//     Standard Inputs/Fix04.N90_STAT/Channel_4/Channel_Error <-> DPO Inputs Channel 4/Channel Error
//     Standard Inputs/Fix04.N90_STAT/Channel_1/Error_Up <-> DPO Inputs Channel 1/Error Up
//     Standard Inputs/Fix04.N90_STAT/Channel_2/Error_Up <-> DPO Inputs Channel 2/Error Up
//     Standard Inputs/Fix04.N90_STAT/Channel_3/Error_Up <-> DPO Inputs Channel 3/Error Up
//     Standard Inputs/Fix04.N90_STAT/Channel_4/Error_Up <-> DPO Inputs Channel 4/Error Up
//     Standard Inputs/Fix04.N90_STAT/Channel_1/Error_Us <-> DPO Inputs Channel 1/Error Us
//     Standard Inputs/Fix04.N90_STAT/Channel_2/Error_Us <-> DPO Inputs Channel 2/Error Us
//     Standard Inputs/Fix04.N90_STAT/Channel_3/Error_Us <-> DPO Inputs Channel 3/Error Us
//     Standard Inputs/Fix04.N90_STAT/Channel_4/Error_Us <-> DPO Inputs Channel 4/Error Us
//     Standard Inputs/Fix04.N90_STAT/Channel_1/Status_Up <-> DPO Inputs Channel 1/Status Up
//     Standard Inputs/Fix04.N90_STAT/Channel_2/Status_Up <-> DPO Inputs Channel 2/Status Up
//     Standard Inputs/Fix04.N90_STAT/Channel_3/Status_Up <-> DPO Inputs Channel 3/Status Up
//     Standard Inputs/Fix04.N90_STAT/Channel_4/Status_Up <-> DPO Inputs Channel 4/Status Up
//     Standard Inputs/Fix04.N90_STAT/Channel_1/Status_Us <-> DPO Inputs Channel 1/Status Us
//     Standard Inputs/Fix04.N90_STAT/Channel_2/Status_Us <-> DPO Inputs Channel 2/Status Us
//     Standard Inputs/Fix04.N90_STAT/Channel_3/Status_Us <-> DPO Inputs Channel 3/Status Us
//     Standard Inputs/Fix04.N90_STAT/Channel_4/Status_Us <-> DPO Inputs Channel 4/Status Us
//     Standard Inputs/Fix04.N90_STAT/Channel_1/SyncError <-> DPO Inputs Channel 1/Sync error
//     Standard Inputs/Fix04.N90_STAT/Channel_2/SyncError <-> DPO Inputs Channel 2/Sync error
//     Standard Inputs/Fix04.N90_STAT/Channel_3/SyncError <-> DPO Inputs Channel 3/Sync error
//     Standard Inputs/Fix04.N90_STAT/Channel_4/SyncError <-> DPO Inputs Channel 4/Sync error
//     Standard Inputs/Fix04.N90_STAT/Channel_1/TxPDO_State <-> DPO Inputs Channel 1/TxPDO State
//     Standard Inputs/Fix04.N90_STAT/Channel_2/TxPDO_State <-> DPO Inputs Channel 2/TxPDO State
//     Standard Inputs/Fix04.N90_STAT/Channel_3/TxPDO_State <-> DPO Inputs Channel 3/TxPDO State
//     Standard Inputs/Fix04.N90_STAT/Channel_4/TxPDO_State <-> DPO Inputs Channel 4/TxPDO State
//     Standard Inputs/Fix04.N90_STAT/Channel_1/TxPDO_Toggle <-> DPO Inputs Channel 1/TxPDO Toggle
//     Standard Inputs/Fix04.N90_STAT/Channel_2/TxPDO_Toggle <-> DPO Inputs Channel 2/TxPDO Toggle
//     Standard Inputs/Fix04.N90_STAT/Channel_3/TxPDO_Toggle <-> DPO Inputs Channel 3/TxPDO Toggle
//     Standard Inputs/Fix04.N90_STAT/Channel_4/TxPDO_Toggle <-> DPO Inputs Channel 4/TxPDO Toggle
//     Standard Inputs/Fix04.N90_STAT/Channel_1/Warning_Up <-> DPO Inputs Channel 1/Warning Up
//     Standard Inputs/Fix04.N90_STAT/Channel_2/Warning_Up <-> DPO Inputs Channel 2/Warning Up
//     Standard Inputs/Fix04.N90_STAT/Channel_3/Warning_Up <-> DPO Inputs Channel 3/Warning Up
//     Standard Inputs/Fix04.N90_STAT/Channel_4/Warning_Up <-> DPO Inputs Channel 4/Warning Up
//     Standard Inputs/Fix04.N90_STAT/Channel_1/Warning_Us <-> DPO Inputs Channel 1/Warning Us
//     Standard Inputs/Fix04.N90_STAT/Channel_2/Warning_Us <-> DPO Inputs Channel 2/Warning Us
//     Standard Inputs/Fix04.N90_STAT/Channel_3/Warning_Us <-> DPO Inputs Channel 3/Warning Us
//     Standard Inputs/Fix04.N90_STAT/Channel_4/Warning_Us <-> DPO Inputs Channel 4/Warning Us
//     Standard Inputs/Fix04.N90_STAT/Device/Global_Error_Bit <-> DPO Inputs Device/Global Error Bit
//     Standard Inputs/Fix04.N90_STAT/Device/Reset_Input <-> DPO Inputs Device/Reset Input
//     Standard Inputs/Fix04.N90_STAT/Device/Temperature_Error <-> DPO Inputs Device/Temperature Error
//     Standard Inputs/Fix04.N90_STAT/Device/Temperature_Warning <-> DPO Inputs Device/Temperature Warning
//     Standard Inputs/Fix04.N90_STAT/Device/TxPDO_State <-> DPO Inputs Device/TxPDO State
//     Standard Inputs/Fix04.N90_STAT/Device/TxPDO_Toggle <-> DPO Inputs Device/TxPDO Toggle
//     Standard Inputs/Fix04.N90_STAT/Device/Up_Error <-> DPO Inputs Device/Up Error
//     Standard Inputs/Fix04.N90_STAT/Device/Up_Warning <-> DPO Inputs Device/Up Warning
//     Standard Inputs/Fix04.N90_STAT/Device/Us_Error <-> DPO Inputs Device/Us Error
//     Standard Inputs/Fix04.N90_STAT/Device/Us_Warning <-> DPO Inputs Device/Us Warning
//     Standard Inputs/Fix04.N90_STAT/InfoData/AdsAddr <-> InfoData/AdsAddr
//     Standard Inputs/Fix04.N90_STAT/InfoData/State <-> InfoData/State
//     Standard Inputs/Fix04.N90_STAT/Wc_State <-> WcState/WcState
//     Standard Outputs/Fix04.N90_CMD/Channel1/Output_Up <-> DPO Outputs Channel 1/Output Up
//     Standard Outputs/Fix04.N90_CMD/Channel2/Output_Up <-> DPO Outputs Channel 2/Output Up
//     Standard Outputs/Fix04.N90_CMD/Channel3/Output_Up <-> DPO Outputs Channel 3/Output Up
//     Standard Outputs/Fix04.N90_CMD/Channel4/Output_Up <-> DPO Outputs Channel 4/Output Up
//     Standard Outputs/Fix04.N90_CMD/Channel1/Output_Us <-> DPO Outputs Channel 1/Output Us
//     Standard Outputs/Fix04.N90_CMD/Channel2/Output_Us <-> DPO Outputs Channel 2/Output Us
//     Standard Outputs/Fix04.N90_CMD/Channel3/Output_Us <-> DPO Outputs Channel 3/Output Us
//     Standard Outputs/Fix04.N90_CMD/Channel4/Output_Us <-> DPO Outputs Channel 4/Output Us
//     Standard Outputs/Fix04.N90_CMD/Channel1/Reset_Up <-> DPO Outputs Channel 1/Reset Up
//     Standard Outputs/Fix04.N90_CMD/Channel2/Reset_Up <-> DPO Outputs Channel 2/Reset Up
//     Standard Outputs/Fix04.N90_CMD/Channel3/Reset_Up <-> DPO Outputs Channel 3/Reset Up
//     Standard Outputs/Fix04.N90_CMD/Channel4/Reset_Up <-> DPO Outputs Channel 4/Reset Up
//     Standard Outputs/Fix04.N90_CMD/Channel1/Reset_Us <-> DPO Outputs Channel 1/Reset Us
//     Standard Outputs/Fix04.N90_CMD/Channel2/Reset_Us <-> DPO Outputs Channel 2/Reset Us
//     Standard Outputs/Fix04.N90_CMD/Channel3/Reset_Us <-> DPO Outputs Channel 3/Reset Us
//     Standard Outputs/Fix04.N90_CMD/Channel4/Reset_Us <-> DPO Outputs Channel 4/Reset Us
//     Standard Outputs/Fix04.N90_CMD/Device/Enable_Control_Via_Fieldbus <-> DPO Outputs Device/Enable Control Via Fieldbus
//     Standard Outputs/Fix04.N90_CMD/Device/Global_Reset <-> DPO Outputs Device/Global Reset
//   SODG11_SSCC610_2403701_PLC/SODG11_SSCC610_2403701_PLC Instance <-> EtherCAT Master (EtherCAT)/IC02.T01 (EK1100)/IC02.T16 (EK1122)/Fix04.N98  (EP2328-0002)
//     Standard Inputs/Fix04.N98.I <-> Channel 1/Input
//     Standard Inputs/Fix04.N98.I @bit 1 <-> Channel 2/Input
//     Standard Inputs/Fix04.N98.I @bit 2 <-> Channel 3/Input
//     Standard Inputs/Fix04.N98.I @bit 3 <-> Channel 4/Input
//     Standard Inputs/Fix04.N98.State <-> InfoData/State
//     Standard Inputs/Fix04.N98.WC_State <-> WcState/WcState
//     Standard Outputs/Fix04.N98.Q <-> Channel 5/Output
//     Standard Outputs/Fix04.N98.Q @bit 1 <-> Channel 6/Output
//     Standard Outputs/Fix04.N98.Q @bit 2 <-> Channel 7/Output
//     Standard Outputs/Fix04.N98.Q @bit 3 <-> Channel 8/Output
//   SODG11_SSCC610_2403701_PLC/SODG11_SSCC610_2403701_PLC Instance <-> EtherCAT Master (EtherCAT)/IC03.T01 (EK1100)
//     Standard Inputs/MAIN.IC03.T01/InfoData/State <-> InfoData/State
//   SODG11_SSCC610_2403701_PLC/SODG11_SSCC610_2403701_PLC Instance <-> EtherCAT Master (EtherCAT)/IC03.T01 (EK1100)/IC03.T02 (EL6900)
//     Standard Inputs/MAIN.IC03.T02_STAT/Device_Info_Data/Project_CRC <-> Device Info Data/Project CRC
//     Standard Inputs/MAIN.IC03.T02_STAT/FBs_FB_ERR <-> StandardInputs/Standard Out Var 26
//     Standard Inputs/MAIN.IC03.T02_STAT/FBs_FB_ERR @bit 8 <-> StandardInputs/Standard Out Var 27
//     Standard Inputs/MAIN.IC03.T02_STAT/FBs_FB_ERR @bit 16 <-> StandardInputs/Standard Out Var 28
//     Standard Inputs/MAIN.IC03.T02_STAT/FBs_FB_ERR @bit 17 <-> StandardInputs/Standard Out Var 29
//     Standard Inputs/MAIN.IC03.T02_STAT/InfoData/AdsAddr/netId <-> InfoData/AdsAddr/netId
//     Standard Inputs/MAIN.IC03.T02_STAT/InfoData/AdsAddr/port <-> InfoData/AdsAddr/port
//     Standard Inputs/MAIN.IC03.T02_STAT/InfoData/State <-> InfoData/State
//     Standard Inputs/MAIN.IC03.T02_STAT/SGs_COM_ERR <-> StandardInputs/Standard Out Var 17
//     Standard Inputs/MAIN.IC03.T02_STAT/SGs_COM_ERR @bit 1 <-> StandardInputs/Standard Out Var 20
//     Standard Inputs/MAIN.IC03.T02_STAT/SGs_FB_ERR <-> StandardInputs/Standard Out Var 16
//     Standard Inputs/MAIN.IC03.T02_STAT/SGs_FB_ERR @bit 1 <-> StandardInputs/Standard Out Var 19
//     Standard Inputs/MAIN.IC03.T02_STAT/SGs_OUT_ERR <-> StandardInputs/Standard Out Var 18
//     Standard Inputs/MAIN.IC03.T02_STAT/SGs_OUT_ERR @bit 1 <-> StandardInputs/Standard Out Var 25
//     Standard Inputs/MAIN.IC03.T09/Q <-> StandardInputs/Standard Out Var 21
//     Standard Inputs/MAIN.IC03.T10/Q <-> StandardInputs/Standard Out Var 23
//     Standard Inputs/MAIN.IC03.T09/Q @bit 1 <-> StandardInputs/Standard Out Var 22
//     Standard Inputs/MAIN.IC03.T10/Q @bit 1 <-> StandardInputs/Standard Out Var 24
//     Standard Outputs/MAIN.IC03.T02_CMD/FBs_ControlPowerPB <-> StandardOutputs/Standard In Var 14
//     Standard Outputs/MAIN.IC03.T02_CMD/SGs_ERRAck <-> StandardOutputs/Standard In Var 11
//     Standard Outputs/MAIN.IC03.T02_CMD/SGs_ERRAck <-> StandardOutputs/Standard In Var 13
//     Standard Outputs/MAIN.IC03.T02_CMD/SGs_RUNSTOP <-> StandardOutputs/Standard In Var 10
//     Standard Outputs/MAIN.IC03.T02_CMD/SGs_RUNSTOP <-> StandardOutputs/Standard In Var 12
//   SODG11_SSCC610_2403701_PLC/SODG11_SSCC610_2403701_PLC Instance <-> EtherCAT Master (EtherCAT)/IC03.T01 (EK1100)/IC03.T03 (EL1904)
//     Standard Inputs/MAIN.IC03.T03/I <-> Module 1 (FSOES)/TxPDO/FSOE/InputChannel1
//     Standard Inputs/MAIN.IC03.T03/I @bit 1 <-> Module 1 (FSOES)/TxPDO/FSOE/InputChannel2
//     Standard Inputs/MAIN.IC03.T03/I @bit 2 <-> Module 1 (FSOES)/TxPDO/FSOE/InputChannel3
//     Standard Inputs/MAIN.IC03.T03/I @bit 3 <-> Module 1 (FSOES)/TxPDO/FSOE/InputChannel4
//     Standard Inputs/MAIN.IC03.T03/InfoData/State <-> InfoData/State
//   SODG11_SSCC610_2403701_PLC/SODG11_SSCC610_2403701_PLC Instance <-> EtherCAT Master (EtherCAT)/IC03.T01 (EK1100)/IC03.T04 (EL1904)
//     Standard Inputs/MAIN.IC03.T04/I <-> Module 1 (FSOES)/TxPDO/FSOE/InputChannel1
//     Standard Inputs/MAIN.IC03.T04/I @bit 1 <-> Module 1 (FSOES)/TxPDO/FSOE/InputChannel2
//     Standard Inputs/MAIN.IC03.T04/I @bit 2 <-> Module 1 (FSOES)/TxPDO/FSOE/InputChannel3
//     Standard Inputs/MAIN.IC03.T04/I @bit 3 <-> Module 1 (FSOES)/TxPDO/FSOE/InputChannel4
//     Standard Inputs/MAIN.IC03.T04/InfoData/State <-> InfoData/State
//   SODG11_SSCC610_2403701_PLC/SODG11_SSCC610_2403701_PLC Instance <-> EtherCAT Master (EtherCAT)/IC03.T01 (EK1100)/IC03.T05 (EL1904)
//     Standard Inputs/MAIN.IC03.T05/I <-> Module 1 (FSOES)/TxPDO/FSOE/InputChannel1
//     Standard Inputs/MAIN.IC03.T05/I @bit 1 <-> Module 1 (FSOES)/TxPDO/FSOE/InputChannel2
//     Standard Inputs/MAIN.IC03.T05/I @bit 2 <-> Module 1 (FSOES)/TxPDO/FSOE/InputChannel3
//     Standard Inputs/MAIN.IC03.T05/I @bit 3 <-> Module 1 (FSOES)/TxPDO/FSOE/InputChannel4
//     Standard Inputs/MAIN.IC03.T05/InfoData/State <-> InfoData/State
//   SODG11_SSCC610_2403701_PLC/SODG11_SSCC610_2403701_PLC Instance <-> EtherCAT Master (EtherCAT)/IC03.T01 (EK1100)/IC03.T06 (EL1904)
//     Standard Inputs/MAIN.IC03.T06/I <-> Module 1 (FSOES)/TxPDO/FSOE/InputChannel1
//     Standard Inputs/MAIN.IC03.T06/I @bit 1 <-> Module 1 (FSOES)/TxPDO/FSOE/InputChannel2
//     Standard Inputs/MAIN.IC03.T06/I @bit 2 <-> Module 1 (FSOES)/TxPDO/FSOE/InputChannel3
//     Standard Inputs/MAIN.IC03.T06/I @bit 3 <-> Module 1 (FSOES)/TxPDO/FSOE/InputChannel4
//     Standard Inputs/MAIN.IC03.T06/InfoData/State <-> InfoData/State
//   SODG11_SSCC610_2403701_PLC/SODG11_SSCC610_2403701_PLC Instance <-> EtherCAT Master (EtherCAT)/IC03.T01 (EK1100)/IC03.T07 (EL1904)
//     Standard Inputs/MAIN.IC03.T07/I <-> Module 1 (FSOES)/TxPDO/FSOE/InputChannel1
//     Standard Inputs/MAIN.IC03.T07/I @bit 1 <-> Module 1 (FSOES)/TxPDO/FSOE/InputChannel2
//     Standard Inputs/MAIN.IC03.T07/I @bit 2 <-> Module 1 (FSOES)/TxPDO/FSOE/InputChannel3
//     Standard Inputs/MAIN.IC03.T07/I @bit 3 <-> Module 1 (FSOES)/TxPDO/FSOE/InputChannel4
//     Standard Inputs/MAIN.IC03.T07/InfoData/State <-> InfoData/State
//   SODG11_SSCC610_2403701_PLC/SODG11_SSCC610_2403701_PLC Instance <-> EtherCAT Master (EtherCAT)/IC03.T01 (EK1100)/IC03.T08 (EL1904)
//     Standard Inputs/MAIN.IC03.T08/I <-> Module 1 (FSOES)/TxPDO/FSOE/InputChannel1
//     Standard Inputs/MAIN.IC03.T08/I @bit 1 <-> Module 1 (FSOES)/TxPDO/FSOE/InputChannel2
//     Standard Inputs/MAIN.IC03.T08/I @bit 2 <-> Module 1 (FSOES)/TxPDO/FSOE/InputChannel3
//     Standard Inputs/MAIN.IC03.T08/I @bit 3 <-> Module 1 (FSOES)/TxPDO/FSOE/InputChannel4
//     Standard Inputs/MAIN.IC03.T08/InfoData/State <-> InfoData/State
//   SODG11_SSCC610_2403701_PLC/SODG11_SSCC610_2403701_PLC Instance <-> EtherCAT Master (EtherCAT)/IC03.T01 (EK1100)/IC03.T09 (EL2904)
//     Standard Inputs/MAIN.IC03.T09/InfoData/State <-> InfoData/State
//   SODG11_SSCC610_2403701_PLC/SODG11_SSCC610_2403701_PLC Instance <-> EtherCAT Master (EtherCAT)/IC03.T01 (EK1100)/IC03.T10 (EL2904)
//     Standard Inputs/MAIN.IC03.T10/InfoData/State <-> InfoData/State
//   SODG11_SSCC610_2403701_PLC/SODG11_SSCC610_2403701_PLC Instance <-> EtherCAT Master (EtherCAT)/IC03.T01 (EK1100)/IC03.T11 (EL9410)
//     Standard Inputs/MAIN.IC03.T11/InfoData/State <-> InfoData/State
//     Standard Inputs/MAIN.IC03.T11/Up_UnderVoltage <-> Status Up/Undervoltage
//     Standard Inputs/MAIN.IC03.T11/Us_Undervoltage <-> Status Us/Undervoltage
//     Standard Inputs/MAIN.IC03.T11/WcState <-> WcState/WcState
//   SODG11_SSCC610_2403701_PLC/SODG11_SSCC610_2403701_PLC Instance <-> EtherCAT Master (EtherCAT)/IC03.T01 (EK1100)/IC03.T12 (EL1004)
//     Standard Inputs/MAIN.IC03.T12/I <-> Channel 1/Input
//     Standard Inputs/MAIN.IC03.T12/I @bit 1 <-> Channel 2/Input
//     Standard Inputs/MAIN.IC03.T12/I @bit 2 <-> Channel 3/Input
//     Standard Inputs/MAIN.IC03.T12/I @bit 3 <-> Channel 4/Input
//     Standard Inputs/MAIN.IC03.T12/InfoData/State <-> InfoData/State
//   SODG11_SSCC610_2403701_PLC/SODG11_SSCC610_2403701_PLC Instance <-> EtherCAT Master (EtherCAT)/IC03.T01 (EK1100)/IC03.T13 (EL1004)
//     Standard Inputs/MAIN.IC03.T13/I <-> Channel 1/Input
//     Standard Inputs/MAIN.IC03.T13/I @bit 1 <-> Channel 2/Input
//     Standard Inputs/MAIN.IC03.T13/I @bit 2 <-> Channel 3/Input
//     Standard Inputs/MAIN.IC03.T13/I @bit 3 <-> Channel 4/Input
//     Standard Inputs/MAIN.IC03.T13/InfoData/State <-> InfoData/State
//   SODG11_SSCC610_2403701_PLC/SODG11_SSCC610_2403701_PLC Instance <-> EtherCAT Master (EtherCAT)/IC03.T01 (EK1100)/IC03.T14 (EL2008)
//     Standard Inputs/MAIN.IC03.T14_STAT/InfoData/State <-> InfoData/State
//     Standard Outputs/MAIN.IC03.T14/Q <-> Channel 1/Output
//     Standard Outputs/MAIN.IC03.T14/Q @bit 1 <-> Channel 2/Output
//     Standard Outputs/MAIN.IC03.T14/Q @bit 2 <-> Channel 3/Output
//     Standard Outputs/MAIN.IC03.T14/Q @bit 3 <-> Channel 4/Output
//     Standard Outputs/MAIN.IC03.T14/Q @bit 4 <-> Channel 5/Output
//     Standard Outputs/MAIN.IC03.T14/Q @bit 5 <-> Channel 6/Output
//     Standard Outputs/MAIN.IC03.T14/Q @bit 6 <-> Channel 7/Output
//     Standard Outputs/MAIN.IC03.T14/Q @bit 7 <-> Channel 8/Output
//   SODG11_SSCC610_2403701_PLC/SODG11_SSCC610_2403701_PLC Instance <-> EtherCAT Master (EtherCAT)/IC03.T01 (EK1100)/IC03.T15 (EL2622)
//     Standard Inputs/MAIN.IC03.T15_STAT/InfoData/State <-> InfoData/State
//     Standard Outputs/MAIN.IC03.T15/Q0 <-> Channel 1/Output
//     Standard Outputs/MAIN.IC03.T15/Q1 <-> Channel 2/Output
//   SODG11_SSCC610_2403701_PLC/SODG11_SSCC610_2403701_PLC Instance <-> EtherCAT Master (EtherCAT)/IC03.T01 (EK1100)/IC03.T16 (EK1122)
//     Standard Inputs/MAIN.IC03.T16/InfoData/State <-> InfoData/State
//   SODG11_SSCC610_2403701_PLC/SODG11_SSCC610_2403701_PLC Instance <-> EtherCAT Master (EtherCAT)/IC03.T01 (EK1100)/IC03.T16 (EK1122)/Fix05.N01 (EP1008-0002)
//     Standard Inputs/Fix05.N01/I <-> Channel 1/Input
//     Standard Inputs/Fix05.N01/I @bit 1 <-> Channel 2/Input
//     Standard Inputs/Fix05.N01/I @bit 2 <-> Channel 3/Input
//     Standard Inputs/Fix05.N01/I @bit 3 <-> Channel 4/Input
//     Standard Inputs/Fix05.N01/I @bit 4 <-> Channel 5/Input
//     Standard Inputs/Fix05.N01/I @bit 5 <-> Channel 6/Input
//     Standard Inputs/Fix05.N01/I @bit 6 <-> Channel 7/Input
//     Standard Inputs/Fix05.N01/I @bit 7 <-> Channel 8/Input
//     Standard Inputs/Fix05.N01/InfoData/State <-> InfoData/State
//     Standard Inputs/Fix05.N01/Wc_State <-> WcState/WcState
//   SODG11_SSCC610_2403701_PLC/SODG11_SSCC610_2403701_PLC Instance <-> EtherCAT Master (EtherCAT)/IC03.T01 (EK1100)/IC03.T16 (EK1122)/Fix05.N02 (EP1008-0002)
//     Standard Inputs/Fix05.N02/I <-> Channel 1/Input
//     Standard Inputs/Fix05.N02/I @bit 1 <-> Channel 2/Input
//     Standard Inputs/Fix05.N02/I @bit 2 <-> Channel 3/Input
//     Standard Inputs/Fix05.N02/I @bit 3 <-> Channel 4/Input
//     Standard Inputs/Fix05.N02/I @bit 4 <-> Channel 5/Input
//     Standard Inputs/Fix05.N02/I @bit 5 <-> Channel 6/Input
//     Standard Inputs/Fix05.N02/I @bit 6 <-> Channel 7/Input
//     Standard Inputs/Fix05.N02/I @bit 7 <-> Channel 8/Input
//     Standard Inputs/Fix05.N02/InfoData/State <-> InfoData/State
//     Standard Inputs/Fix05.N02/Wc_State <-> WcState/WcState
//   SODG11_SSCC610_2403701_PLC/SODG11_SSCC610_2403701_PLC Instance <-> EtherCAT Master (EtherCAT)/IC03.T01 (EK1100)/IC03.T16 (EK1122)/Fix05.N03 (EP1008-0002)
//     Standard Inputs/Fix05.N03/I <-> Channel 1/Input
//     Standard Inputs/Fix05.N03/I @bit 1 <-> Channel 2/Input
//     Standard Inputs/Fix05.N03/I @bit 2 <-> Channel 3/Input
//     Standard Inputs/Fix05.N03/I @bit 3 <-> Channel 4/Input
//     Standard Inputs/Fix05.N03/I @bit 4 <-> Channel 5/Input
//     Standard Inputs/Fix05.N03/I @bit 5 <-> Channel 6/Input
//     Standard Inputs/Fix05.N03/I @bit 6 <-> Channel 7/Input
//     Standard Inputs/Fix05.N03/I @bit 7 <-> Channel 8/Input
//     Standard Inputs/Fix05.N03/InfoData/State <-> InfoData/State
//     Standard Inputs/Fix05.N03/Wc_State <-> WcState/WcState
//   SODG11_SSCC610_2403701_PLC/SODG11_SSCC610_2403701_PLC Instance <-> EtherCAT Master (EtherCAT)/IC03.T01 (EK1100)/IC03.T16 (EK1122)/Fix05.N04 (EP1008-0002)
//     Standard Inputs/Fix05.N04/I <-> Channel 1/Input
//     Standard Inputs/Fix05.N04/I @bit 1 <-> Channel 2/Input
//     Standard Inputs/Fix05.N04/I @bit 2 <-> Channel 3/Input
//     Standard Inputs/Fix05.N04/I @bit 3 <-> Channel 4/Input
//     Standard Inputs/Fix05.N04/I @bit 4 <-> Channel 5/Input
//     Standard Inputs/Fix05.N04/I @bit 5 <-> Channel 6/Input
//     Standard Inputs/Fix05.N04/I @bit 6 <-> Channel 7/Input
//     Standard Inputs/Fix05.N04/I @bit 7 <-> Channel 8/Input
//     Standard Inputs/Fix05.N04/InfoData/State <-> InfoData/State
//     Standard Inputs/Fix05.N04/Wc_State <-> WcState/WcState
//   SODG11_SSCC610_2403701_PLC/SODG11_SSCC610_2403701_PLC Instance <-> EtherCAT Master (EtherCAT)/IC03.T01 (EK1100)/IC03.T16 (EK1122)/Fix05.N100 (EX260-SEC1)
//     Standard Inputs/Fix05.N100_STAT/InfoData/State <-> InfoData/State
//     Standard Outputs/Fix05.N100/Q <-> Byte 0/Output
//     Standard Outputs/Fix05.N100/Q @bit 8 <-> Byte 1/Output
//     Standard Outputs/Fix05.N100/Q @bit 16 <-> Byte 2/Output
//     Standard Outputs/Fix05.N100/Q @bit 24 <-> Byte 3/Output
//   SODG11_SSCC610_2403701_PLC/SODG11_SSCC610_2403701_PLC Instance <-> EtherCAT Master (EtherCAT)/IC03.T01 (EK1100)/IC03.T16 (EK1122)/Fix102.N01 (EP1008-0002)
//     Standard Inputs/Fix102.N01/I <-> Channel 1/Input
//     Standard Inputs/Fix102.N01/I @bit 1 <-> Channel 2/Input
//     Standard Inputs/Fix102.N01/I @bit 2 <-> Channel 3/Input
//     Standard Inputs/Fix102.N01/I @bit 3 <-> Channel 4/Input
//     Standard Inputs/Fix102.N01/I @bit 4 <-> Channel 5/Input
//     Standard Inputs/Fix102.N01/I @bit 5 <-> Channel 6/Input
//     Standard Inputs/Fix102.N01/I @bit 6 <-> Channel 7/Input
//     Standard Inputs/Fix102.N01/I @bit 7 <-> Channel 8/Input
//     Standard Inputs/Fix102.N01/InfoData/State <-> InfoData/State
//     Standard Inputs/Fix102.N01/Wc_State <-> WcState/WcState
//   SODG11_SSCC610_2403701_PLC/SODG11_SSCC610_2403701_PLC Instance <-> EtherCAT Master (EtherCAT)/IC03.T01 (EK1100)/IC03.T16 (EK1122)/Fix102.N02 (EP1008-0002)
//     Standard Inputs/Fix102.N02/I <-> Channel 1/Input
//     Standard Inputs/Fix102.N02/I @bit 1 <-> Channel 2/Input
//     Standard Inputs/Fix102.N02/I @bit 2 <-> Channel 3/Input
//     Standard Inputs/Fix102.N02/I @bit 3 <-> Channel 4/Input
//     Standard Inputs/Fix102.N02/I @bit 4 <-> Channel 5/Input
//     Standard Inputs/Fix102.N02/I @bit 5 <-> Channel 6/Input
//     Standard Inputs/Fix102.N02/I @bit 6 <-> Channel 7/Input
//     Standard Inputs/Fix102.N02/I @bit 7 <-> Channel 8/Input
//     Standard Inputs/Fix102.N02/InfoData/State <-> InfoData/State
//     Standard Inputs/Fix102.N02/Wc_State <-> WcState/WcState
//   SODG11_SSCC610_2403701_PLC/SODG11_SSCC610_2403701_PLC Instance <-> EtherCAT Master (EtherCAT)/IC03.T01 (EK1100)/IC03.T16 (EK1122)/Fix102.N03 (EP1008-0002)
//     Standard Inputs/Fix102.N03/I <-> Channel 1/Input
//     Standard Inputs/Fix102.N03/I @bit 1 <-> Channel 2/Input
//     Standard Inputs/Fix102.N03/I @bit 2 <-> Channel 3/Input
//     Standard Inputs/Fix102.N03/I @bit 3 <-> Channel 4/Input
//     Standard Inputs/Fix102.N03/I @bit 4 <-> Channel 5/Input
//     Standard Inputs/Fix102.N03/I @bit 5 <-> Channel 6/Input
//     Standard Inputs/Fix102.N03/I @bit 6 <-> Channel 7/Input
//     Standard Inputs/Fix102.N03/I @bit 7 <-> Channel 8/Input
//     Standard Inputs/Fix102.N03/InfoData/State <-> InfoData/State
//     Standard Inputs/Fix102.N03/Wc_State <-> WcState/WcState
//   SODG11_SSCC610_2403701_PLC/SODG11_SSCC610_2403701_PLC Instance <-> EtherCAT Master (EtherCAT)/IC03.T01 (EK1100)/IC03.T16 (EK1122)/Fix102.N04 (EP1008-0002)
//     Standard Inputs/Fix102.N04/I <-> Channel 1/Input
//     Standard Inputs/Fix102.N04/I @bit 1 <-> Channel 2/Input
//     Standard Inputs/Fix102.N04/I @bit 2 <-> Channel 3/Input
//     Standard Inputs/Fix102.N04/I @bit 3 <-> Channel 4/Input
//     Standard Inputs/Fix102.N04/I @bit 4 <-> Channel 5/Input
//     Standard Inputs/Fix102.N04/I @bit 5 <-> Channel 6/Input
//     Standard Inputs/Fix102.N04/I @bit 6 <-> Channel 7/Input
//     Standard Inputs/Fix102.N04/I @bit 7 <-> Channel 8/Input
//     Standard Inputs/Fix102.N04/InfoData/State <-> InfoData/State
//     Standard Inputs/Fix102.N04/Wc_State <-> WcState/WcState
//   SODG11_SSCC610_2403701_PLC/SODG11_SSCC610_2403701_PLC Instance <-> EtherCAT Master (EtherCAT)/IC03.T01 (EK1100)/IC03.T16 (EK1122)/Fix102.N100 (EX260-SEC1)
//     Standard Inputs/Fix102.N100_STAT/InfoData/State <-> InfoData/State
//     Standard Outputs/Fix102.N100/Q <-> Byte 0/Output
//     Standard Outputs/Fix102.N100/Q @bit 8 <-> Byte 1/Output
//     Standard Outputs/Fix102.N100/Q @bit 16 <-> Byte 2/Output
//     Standard Outputs/Fix102.N100/Q @bit 24 <-> Byte 3/Output
//   SODG11_SSCC610_2403701_PLC/SODG11_SSCC610_2403701_PLC Instance <-> EtherCAT Master (EtherCAT)/IC03.T01 (EK1100)/IC03.T16 (EK1122)/QA_Fix102CAM1 (DL-EC1A)
//     Standard Inputs/Fix102.QA_IV3[1].ECAT_Input_Data/Busy <-> ID06 Status/Busy
//     Standard Inputs/Fix102.QA_IV3[1].ECAT_Input_Data/ErrorClearResponse <-> ID06 Status/Clear Error Ack
//     Standard Inputs/Fix102.QA_IV3[1].ECAT_Input_Data/ErrorCode <-> Status of System/Error Code
//     Standard Inputs/Fix102.QA_IV3[1].ECAT_Input_Data/Error_Status <-> Status of System/Error Status
//     Standard Inputs/Fix102.QA_IV3[1].ECAT_Input_Data/InfoData/State <-> InfoData/State
//     Standard Inputs/Fix102.QA_IV3[1].ECAT_Input_Data/LogicResult[1] <-> ID04 Status/Logic 01
//     Standard Inputs/Fix102.QA_IV3[1].ECAT_Input_Data/LogicResult[2] <-> ID05 Status/Logic 02
//     Standard Inputs/Fix102.QA_IV3[1].ECAT_Input_Data/LogicResult[3] <-> ID06 Status/Logic 03
//     Standard Inputs/Fix102.QA_IV3[1].ECAT_Input_Data/LogicResult[4] <-> ID07 Status/Logic 04
//     Standard Inputs/Fix102.QA_IV3[1].ECAT_Input_Data/MasterRegFailed <-> ID03 Status/Regist Master Image Failed
//     Standard Inputs/Fix102.QA_IV3[1].ECAT_Input_Data/MasterRegResponse <-> ID03 Status/Regist Master Image Ack
//     Standard Inputs/Fix102.QA_IV3[1].ECAT_Input_Data/NoFreeSpaceSD <-> ID08 Status/SD Card No Space
//     Standard Inputs/Fix102.QA_IV3[1].ECAT_Input_Data/OverallJudgementOK <-> ID01 Status/Total Status OK
//     Standard Inputs/Fix102.QA_IV3[1].ECAT_Input_Data/PositionAdjMatch <-> ID02 Current Value/Tool 00 Score
//     Standard Inputs/Fix102.QA_IV3[1].ECAT_Input_Data/PositionCorrectionStatus <-> ID02 Status/Tool 00 Status
//     Standard Inputs/Fix102.QA_IV3[1].ECAT_Input_Data/ProgramNumber <-> ID01 Status/Program Num 00
//     Standard Inputs/Fix102.QA_IV3[1].ECAT_Input_Data/ProgramNumber @bit 1 <-> ID02 Status/Program Num 01
//     Standard Inputs/Fix102.QA_IV3[1].ECAT_Input_Data/ProgramNumber @bit 2 <-> ID03 Status/Program Num 02
//     Standard Inputs/Fix102.QA_IV3[1].ECAT_Input_Data/ProgramNumber @bit 3 <-> ID04 Status/Program Num 03
//     Standard Inputs/Fix102.QA_IV3[1].ECAT_Input_Data/ProgramNumber @bit 4 <-> ID05 Status/Program Num 04
//     Standard Inputs/Fix102.QA_IV3[1].ECAT_Input_Data/ProgramNumber @bit 5 <-> ID06 Status/Program Num 05
//     Standard Inputs/Fix102.QA_IV3[1].ECAT_Input_Data/ProgramNumber @bit 6 <-> ID07 Status/Program Num 06
//     Standard Inputs/Fix102.QA_IV3[1].ECAT_Input_Data/ProgramSwitchFailed <-> ID01 Status/Change Program Failed
//     Standard Inputs/Fix102.QA_IV3[1].ECAT_Input_Data/ProgramSwitchOK <-> ID01 Status/Change Program Ack
//     Standard Inputs/Fix102.QA_IV3[1].ECAT_Input_Data/ResultAvailable <-> ID01 Status/Result Valid
//     Standard Inputs/Fix102.QA_IV3[1].ECAT_Input_Data/ResultUpdateComplete <-> ID02 Status/Result Updated Toggle
//     Standard Inputs/Fix102.QA_IV3[1].ECAT_Input_Data/Running <-> ID05 Status/Run
//     Standard Inputs/Fix102.QA_IV3[1].ECAT_Input_Data/SDCardStopFailed <-> ID04 Status/SD Card Detected
//     Standard Inputs/Fix102.QA_IV3[1].ECAT_Input_Data/SDCardStopResponse <-> ID04 Status/SD Save Stop Ack
//     Standard Inputs/Fix102.QA_IV3[1].ECAT_Input_Data/StatsResetResponse <-> ID05 Status/Reset Statistics Ack
//     Standard Inputs/Fix102.QA_IV3[1].ECAT_Input_Data/ToolMatch[10] <-> ID12 Current Value/Tool 10 Score
//     Standard Inputs/Fix102.QA_IV3[1].ECAT_Input_Data/ToolMatch[11] <-> ID13 Current Value/Tool 11 Score
//     Standard Inputs/Fix102.QA_IV3[1].ECAT_Input_Data/ToolMatch[12] <-> ID14 Current Value/Tool 12 Score
//     Standard Inputs/Fix102.QA_IV3[1].ECAT_Input_Data/ToolMatch[13] <-> ID15 Current Value/Tool 13 Score
//     Standard Inputs/Fix102.QA_IV3[1].ECAT_Input_Data/ToolMatch[1] <-> ID03 Current Value/Tool 01 Score
//     Standard Inputs/Fix102.QA_IV3[1].ECAT_Input_Data/ToolMatch[2] <-> ID04 Current Value/Tool 02 Score
//     Standard Inputs/Fix102.QA_IV3[1].ECAT_Input_Data/ToolMatch[3] <-> ID05 Current Value/Tool 03 Score
//     Standard Inputs/Fix102.QA_IV3[1].ECAT_Input_Data/ToolMatch[4] <-> ID06 Current Value/Tool 04 Score
//     Standard Inputs/Fix102.QA_IV3[1].ECAT_Input_Data/ToolMatch[5] <-> ID07 Current Value/Tool 05 Score
//     Standard Inputs/Fix102.QA_IV3[1].ECAT_Input_Data/ToolMatch[6] <-> ID08 Current Value/Tool 06 Score
//     Standard Inputs/Fix102.QA_IV3[1].ECAT_Input_Data/ToolMatch[7] <-> ID09 Current Value/Tool 07 Score
//     Standard Inputs/Fix102.QA_IV3[1].ECAT_Input_Data/ToolMatch[8] <-> ID10 Current Value/Tool 08 Score
//     Standard Inputs/Fix102.QA_IV3[1].ECAT_Input_Data/ToolMatch[9] <-> ID11 Current Value/Tool 09 Score
//     Standard Inputs/Fix102.QA_IV3[1].ECAT_Input_Data/ToolResult[10] <-> ID12 Status/Tool 10 Status
//     Standard Inputs/Fix102.QA_IV3[1].ECAT_Input_Data/ToolResult[11] <-> ID13 Status/Tool 11 Status
//     Standard Inputs/Fix102.QA_IV3[1].ECAT_Input_Data/ToolResult[12] <-> ID14 Status/Tool 12 Status
//     Standard Inputs/Fix102.QA_IV3[1].ECAT_Input_Data/ToolResult[13] <-> ID15 Status/Tool 13 Status
//     Standard Inputs/Fix102.QA_IV3[1].ECAT_Input_Data/ToolResult[1] <-> ID03 Status/Tool 01 Status
//     Standard Inputs/Fix102.QA_IV3[1].ECAT_Input_Data/ToolResult[2] <-> ID04 Status/Tool 02 Status
//     Standard Inputs/Fix102.QA_IV3[1].ECAT_Input_Data/ToolResult[3] <-> ID05 Status/Tool 03 Status
//     Standard Inputs/Fix102.QA_IV3[1].ECAT_Input_Data/ToolResult[4] <-> ID06 Status/Tool 04 Status
//     Standard Inputs/Fix102.QA_IV3[1].ECAT_Input_Data/ToolResult[5] <-> ID07 Status/Tool 05 Status
//     Standard Inputs/Fix102.QA_IV3[1].ECAT_Input_Data/ToolResult[6] <-> ID08 Status/Tool 06 Status
//     Standard Inputs/Fix102.QA_IV3[1].ECAT_Input_Data/ToolResult[7] <-> ID09 Status/Tool 07 Status
//     Standard Inputs/Fix102.QA_IV3[1].ECAT_Input_Data/ToolResult[8] <-> ID10 Status/Tool 08 Status
//     Standard Inputs/Fix102.QA_IV3[1].ECAT_Input_Data/ToolResult[9] <-> ID11 Status/Tool 09 Status
//     Standard Inputs/Fix102.QA_IV3[1].ECAT_Input_Data/TriggerFailed <-> ID02 Status/Trigger Failed
//     Standard Inputs/Fix102.QA_IV3[1].ECAT_Input_Data/TriggerReady <-> ID07 Status/Trigger Ready
//     Standard Inputs/Fix102.QA_IV3[1].ECAT_Input_Data/TriggerResponse <-> ID02 Status/Trigger Ack
//     Standard Outputs/Fix102.QA_IV3[1].ECAT_Output_Data[{1..5}] <-> Input Request {1..5}/Request {1..5}  (5 links)
//   SODG11_SSCC610_2403701_PLC/SODG11_SSCC610_2403701_PLC Instance <-> EtherCAT Master (EtherCAT)/IC03.T01 (EK1100)/IC03.T16 (EK1122)/QA_Fix102CAM2 (DL-EC1A)
//     Standard Inputs/Fix102.QA_IV3[2].ECAT_Input_Data/Busy <-> ID06 Status/Busy
//     Standard Inputs/Fix102.QA_IV3[2].ECAT_Input_Data/ErrorClearResponse <-> ID06 Status/Clear Error Ack
//     Standard Inputs/Fix102.QA_IV3[2].ECAT_Input_Data/ErrorCode <-> Status of System/Error Code
//     Standard Inputs/Fix102.QA_IV3[2].ECAT_Input_Data/Error_Status <-> Status of System/Error Status
//     Standard Inputs/Fix102.QA_IV3[2].ECAT_Input_Data/InfoData/State <-> InfoData/State
//     Standard Inputs/Fix102.QA_IV3[2].ECAT_Input_Data/LogicResult[1] <-> ID04 Status/Logic 01
//     Standard Inputs/Fix102.QA_IV3[2].ECAT_Input_Data/LogicResult[2] <-> ID05 Status/Logic 02
//     Standard Inputs/Fix102.QA_IV3[2].ECAT_Input_Data/LogicResult[3] <-> ID06 Status/Logic 03
//     Standard Inputs/Fix102.QA_IV3[2].ECAT_Input_Data/LogicResult[4] <-> ID07 Status/Logic 04
//     Standard Inputs/Fix102.QA_IV3[2].ECAT_Input_Data/MasterRegFailed <-> ID03 Status/Regist Master Image Failed
//     Standard Inputs/Fix102.QA_IV3[2].ECAT_Input_Data/MasterRegResponse <-> ID03 Status/Regist Master Image Ack
//     Standard Inputs/Fix102.QA_IV3[2].ECAT_Input_Data/NoFreeSpaceSD <-> ID08 Status/SD Card No Space
//     Standard Inputs/Fix102.QA_IV3[2].ECAT_Input_Data/OverallJudgementOK <-> ID01 Status/Total Status OK
//     Standard Inputs/Fix102.QA_IV3[2].ECAT_Input_Data/PositionAdjMatch <-> ID02 Current Value/Tool 00 Score
//     Standard Inputs/Fix102.QA_IV3[2].ECAT_Input_Data/PositionCorrectionStatus <-> ID02 Status/Tool 00 Status
//     Standard Inputs/Fix102.QA_IV3[2].ECAT_Input_Data/ProgramNumber <-> ID01 Status/Program Num 00
//     Standard Inputs/Fix102.QA_IV3[2].ECAT_Input_Data/ProgramNumber @bit 1 <-> ID02 Status/Program Num 01
//     Standard Inputs/Fix102.QA_IV3[2].ECAT_Input_Data/ProgramNumber @bit 2 <-> ID03 Status/Program Num 02
//     Standard Inputs/Fix102.QA_IV3[2].ECAT_Input_Data/ProgramNumber @bit 3 <-> ID04 Status/Program Num 03
//     Standard Inputs/Fix102.QA_IV3[2].ECAT_Input_Data/ProgramNumber @bit 4 <-> ID05 Status/Program Num 04
//     Standard Inputs/Fix102.QA_IV3[2].ECAT_Input_Data/ProgramNumber @bit 5 <-> ID06 Status/Program Num 05
//     Standard Inputs/Fix102.QA_IV3[2].ECAT_Input_Data/ProgramNumber @bit 6 <-> ID07 Status/Program Num 06
//     Standard Inputs/Fix102.QA_IV3[2].ECAT_Input_Data/ProgramSwitchFailed <-> ID01 Status/Change Program Failed
//     Standard Inputs/Fix102.QA_IV3[2].ECAT_Input_Data/ProgramSwitchOK <-> ID01 Status/Change Program Ack
//     Standard Inputs/Fix102.QA_IV3[2].ECAT_Input_Data/ResultAvailable <-> ID01 Status/Result Valid
//     Standard Inputs/Fix102.QA_IV3[2].ECAT_Input_Data/ResultUpdateComplete <-> ID02 Status/Result Updated Toggle
//     Standard Inputs/Fix102.QA_IV3[2].ECAT_Input_Data/Running <-> ID05 Status/Run
//     Standard Inputs/Fix102.QA_IV3[2].ECAT_Input_Data/SDCardStopFailed <-> ID04 Status/SD Card Detected
//     Standard Inputs/Fix102.QA_IV3[2].ECAT_Input_Data/SDCardStopResponse <-> ID04 Status/SD Save Stop Ack
//     Standard Inputs/Fix102.QA_IV3[2].ECAT_Input_Data/StatsResetResponse <-> ID05 Status/Reset Statistics Ack
//     Standard Inputs/Fix102.QA_IV3[2].ECAT_Input_Data/ToolMatch[10] <-> ID12 Current Value/Tool 10 Score
//     Standard Inputs/Fix102.QA_IV3[2].ECAT_Input_Data/ToolMatch[11] <-> ID13 Current Value/Tool 11 Score
//     Standard Inputs/Fix102.QA_IV3[2].ECAT_Input_Data/ToolMatch[12] <-> ID14 Current Value/Tool 12 Score
//     Standard Inputs/Fix102.QA_IV3[2].ECAT_Input_Data/ToolMatch[13] <-> ID15 Current Value/Tool 13 Score
//     Standard Inputs/Fix102.QA_IV3[2].ECAT_Input_Data/ToolMatch[1] <-> ID03 Current Value/Tool 01 Score
//     Standard Inputs/Fix102.QA_IV3[2].ECAT_Input_Data/ToolMatch[2] <-> ID04 Current Value/Tool 02 Score
//     Standard Inputs/Fix102.QA_IV3[2].ECAT_Input_Data/ToolMatch[3] <-> ID05 Current Value/Tool 03 Score
//     Standard Inputs/Fix102.QA_IV3[2].ECAT_Input_Data/ToolMatch[4] <-> ID06 Current Value/Tool 04 Score
//     Standard Inputs/Fix102.QA_IV3[2].ECAT_Input_Data/ToolMatch[5] <-> ID07 Current Value/Tool 05 Score
//     Standard Inputs/Fix102.QA_IV3[2].ECAT_Input_Data/ToolMatch[6] <-> ID08 Current Value/Tool 06 Score
//     Standard Inputs/Fix102.QA_IV3[2].ECAT_Input_Data/ToolMatch[7] <-> ID09 Current Value/Tool 07 Score
//     Standard Inputs/Fix102.QA_IV3[2].ECAT_Input_Data/ToolMatch[8] <-> ID10 Current Value/Tool 08 Score
//     Standard Inputs/Fix102.QA_IV3[2].ECAT_Input_Data/ToolMatch[9] <-> ID11 Current Value/Tool 09 Score
//     Standard Inputs/Fix102.QA_IV3[2].ECAT_Input_Data/ToolResult[10] <-> ID12 Status/Tool 10 Status
//     Standard Inputs/Fix102.QA_IV3[2].ECAT_Input_Data/ToolResult[11] <-> ID13 Status/Tool 11 Status
//     Standard Inputs/Fix102.QA_IV3[2].ECAT_Input_Data/ToolResult[12] <-> ID14 Status/Tool 12 Status
//     Standard Inputs/Fix102.QA_IV3[2].ECAT_Input_Data/ToolResult[13] <-> ID15 Status/Tool 13 Status
//     Standard Inputs/Fix102.QA_IV3[2].ECAT_Input_Data/ToolResult[1] <-> ID03 Status/Tool 01 Status
//     Standard Inputs/Fix102.QA_IV3[2].ECAT_Input_Data/ToolResult[2] <-> ID04 Status/Tool 02 Status
//     Standard Inputs/Fix102.QA_IV3[2].ECAT_Input_Data/ToolResult[3] <-> ID05 Status/Tool 03 Status
//     Standard Inputs/Fix102.QA_IV3[2].ECAT_Input_Data/ToolResult[4] <-> ID06 Status/Tool 04 Status
//     Standard Inputs/Fix102.QA_IV3[2].ECAT_Input_Data/ToolResult[5] <-> ID07 Status/Tool 05 Status
//     Standard Inputs/Fix102.QA_IV3[2].ECAT_Input_Data/ToolResult[6] <-> ID08 Status/Tool 06 Status
//     Standard Inputs/Fix102.QA_IV3[2].ECAT_Input_Data/ToolResult[7] <-> ID09 Status/Tool 07 Status
//     Standard Inputs/Fix102.QA_IV3[2].ECAT_Input_Data/ToolResult[8] <-> ID10 Status/Tool 08 Status
//     Standard Inputs/Fix102.QA_IV3[2].ECAT_Input_Data/ToolResult[9] <-> ID11 Status/Tool 09 Status
//     Standard Inputs/Fix102.QA_IV3[2].ECAT_Input_Data/TriggerFailed <-> ID02 Status/Trigger Failed
//     Standard Inputs/Fix102.QA_IV3[2].ECAT_Input_Data/TriggerReady <-> ID07 Status/Trigger Ready
//     Standard Inputs/Fix102.QA_IV3[2].ECAT_Input_Data/TriggerResponse <-> ID02 Status/Trigger Ack
//     Standard Outputs/Fix102.QA_IV3[2].ECAT_Output_Data[{1..5}] <-> Input Request {1..5}/Request {1..5}  (5 links)
//   SODG11_SSCC610_2403701_PLC/SODG11_SSCC610_2403701_PLC Instance <-> EtherCAT Master (EtherCAT)/IS01.T01 (EK1100)
//     Standard Inputs/MAIN.IS01.T01/InfoData/State <-> InfoData/State
//   SODG11_SSCC610_2403701_PLC/SODG11_SSCC610_2403701_PLC Instance <-> EtherCAT Master (EtherCAT)/IS01.T01 (EK1100)/IS01.T02 (EL6900)
//     Standard Inputs/MAIN.IS01.T02_STAT/Device_Info_Data/Project_CRC <-> Device Info Data/Project CRC
//     Standard Inputs/MAIN.IS01.T02_STAT/InfoData/State <-> InfoData/State
//     Standard Inputs/MAIN.IS01.T02_STAT/SGs_COM_ERR @bit 1 <-> StandardInputs/Standard Out Var 12
//     Standard Inputs/MAIN.IS01.T02_STAT/SGs_COM_ERR <-> StandardInputs/Standard Out Var 9
//     Standard Inputs/MAIN.IS01.T02_STAT/SGs_FB_ERR @bit 1 <-> StandardInputs/Standard Out Var 11
//     Standard Inputs/MAIN.IS01.T02_STAT/SGs_FB_ERR <-> StandardInputs/Standard Out Var 8
//     Standard Inputs/MAIN.IS01.T02_STAT/SGs_OUT_ERR <-> StandardInputs/Standard Out Var 10
//     Standard Inputs/MAIN.IS01.T02_STAT/SGs_OUT_ERR @bit 1 <-> StandardInputs/Standard Out Var 13
//     Standard Inputs/MAIN.IS01.T04/Q <-> StandardInputs/Standard Out Var 14
//     Standard Inputs/MAIN.IS01.T04/Q @bit 1 <-> StandardInputs/Standard Out Var 15
//     Standard Inputs/MAIN.IS01.T04/Q @bit 2 <-> StandardInputs/Standard Out Var 16
//     Standard Inputs/MAIN.IS01.T04/Q @bit 3 <-> StandardInputs/Standard Out Var 17
//     Standard Outputs/MAIN.IS01.T02_CMD/SGs_ERRAck <-> StandardOutputs/Standard In Var 5
//     Standard Outputs/MAIN.IS01.T02_CMD/SGs_ERRAck <-> StandardOutputs/Standard In Var 7
//     Standard Outputs/MAIN.IS01.T02_CMD/SGs_RUNSTOP <-> StandardOutputs/Standard In Var 4
//     Standard Outputs/MAIN.IS01.T02_CMD/SGs_RUNSTOP <-> StandardOutputs/Standard In Var 6
//   SODG11_SSCC610_2403701_PLC/SODG11_SSCC610_2403701_PLC Instance <-> EtherCAT Master (EtherCAT)/IS01.T01 (EK1100)/IS01.T03 (EL1904)
//     Standard Inputs/MAIN.IS01.T03/I <-> Module 1 (FSOES)/TxPDO/FSOE/InputChannel1
//     Standard Inputs/MAIN.IS01.T03/I @bit 1 <-> Module 1 (FSOES)/TxPDO/FSOE/InputChannel2
//     Standard Inputs/MAIN.IS01.T03/I @bit 2 <-> Module 1 (FSOES)/TxPDO/FSOE/InputChannel3
//     Standard Inputs/MAIN.IS01.T03/I @bit 3 <-> Module 1 (FSOES)/TxPDO/FSOE/InputChannel4
//     Standard Inputs/MAIN.IS01.T03/InfoData/State <-> InfoData/State
//   SODG11_SSCC610_2403701_PLC/SODG11_SSCC610_2403701_PLC Instance <-> EtherCAT Master (EtherCAT)/IS01.T01 (EK1100)/IS01.T04 (EL2904)
//     Standard Inputs/MAIN.IS01.T04/InfoData/State <-> InfoData/State
//   SODG11_SSCC610_2403701_PLC/SODG11_SSCC610_2403701_PLC Instance <-> EtherCAT Master (EtherCAT)/IS01.T01 (EK1100)/IS01.T05 (EL6731)
//     Standard Inputs/MAIN.IS01.T05/InfoData/State <-> InfoData/State
//   SODG11_SSCC610_2403701_PLC/SODG11_SSCC610_2403701_PLC Instance <-> EtherCAT Master (EtherCAT)/IS01.T01 (EK1100)/IS01.T06 (EK1110)
//     Standard Inputs/MAIN.IS01.T06/InfoData/State <-> InfoData/State
//   SODG11_SSCC610_2403701_PLC/SODG11_SSCC610_2403701_PLC Instance <-> EtherCAT Master (EtherCAT)/MD01.N01 (EP1918-0002)
//     Standard Inputs/MAIN.MD01.N01_STAT/Device_Info_Data/Project_CRC <-> Device Info Data/Project CRC
//     Standard Inputs/MAIN.MD01.N01_STAT/FBs_FB_ERR @bit 8 <-> StandardInputs/Standard Out Var 13
//     Standard Inputs/MAIN.MD01.N01_STAT/InfoData/AdsAddr/netId <-> InfoData/AdsAddr/netId
//     Standard Inputs/MAIN.MD01.N01_STAT/InfoData/AdsAddr/port <-> InfoData/AdsAddr/port
//     Standard Inputs/MAIN.MD01.N01_STAT/InfoData/State <-> InfoData/State
//     Standard Inputs/MAIN.MD01.N01_STAT/SGs_COM_ERR @bit 1 <-> StandardInputs/Standard Out Var 24
//     Standard Inputs/MAIN.MD01.N01_STAT/SGs_COM_ERR <-> StandardInputs/Standard Out Var 9
//     Standard Inputs/MAIN.MD01.N01_STAT/SGs_FB_ERR <-> StandardInputs/Standard Out Var 10
//     Standard Inputs/MAIN.MD01_N01_I0 <-> StandardInputs/Standard Out Var 34
//     Standard Inputs/MAIN.MD01_N01_I1 <-> StandardInputs/Standard Out Var 35
//     Standard Inputs/MAIN.MD01_N01_I2 <-> StandardInputs/Standard Out Var 36
//     Standard Inputs/MAIN.MD01_N01_I3 <-> StandardInputs/Standard Out Var 37
//     Standard Outputs/MAIN.MD01.N01_CMD/FBs_Restart_Spare <-> StandardOutputs/Standard In Var 23
//     Standard Outputs/MAIN.MD01.N01_CMD/SGs_ERRAck <-> StandardOutputs/Standard In Var 1
//     Standard Outputs/MAIN.MD01.N01_CMD/SGs_RUNSTOP <-> StandardOutputs/Standard In Var 2
//   SODG11_SSCC610_2403701_PLC/SODG11_SSCC610_2403701_PLC Instance <-> EtherCAT Master (EtherCAT)/MD01.N02 (EP1008-0002)
//     Standard Inputs/MAIN.MD01.N02/I <-> Channel 1/Input
//     Standard Inputs/MAIN.MD01.N02/I @bit 1 <-> Channel 2/Input
//     Standard Inputs/MAIN.MD01.N02/I @bit 2 <-> Channel 3/Input
//     Standard Inputs/MAIN.MD01.N02/I @bit 3 <-> Channel 4/Input
//     Standard Inputs/MAIN.MD01.N02/I @bit 4 <-> Channel 5/Input
//     Standard Inputs/MAIN.MD01.N02/I @bit 5 <-> Channel 6/Input
//     Standard Inputs/MAIN.MD01.N02/I @bit 6 <-> Channel 7/Input
//     Standard Inputs/MAIN.MD01.N02/I @bit 7 <-> Channel 8/Input
//     Standard Inputs/MAIN.MD01.N02/InfoData/State <-> InfoData/State
//   SODG11_SSCC610_2403701_PLC/SODG11_SSCC610_2403701_PLC Instance <-> EtherCAT Master (EtherCAT)/MD01.N03 (EP2624-0002)
//     Standard Inputs/MAIN.MD01.N03_STAT/InfoData/State <-> InfoData/State
//     Standard Outputs/MAIN.MD01.N03/Q <-> Channel 1/Output
//     Standard Outputs/MAIN.MD01.N03/Q @bit 1 <-> Channel 2/Output
//     Standard Outputs/MAIN.MD01.N03/Q @bit 2 <-> Channel 3/Output
//     Standard Outputs/MAIN.MD01.N03/Q @bit 3 <-> Channel 4/Output
//   SODG11_SSCC610_2403701_PLC/SODG11_SSCC610_2403701_PLC Instance <-> EtherCAT Master (EtherCAT)/MD02.N01 (EP1918-0002)
//     Standard Inputs/MAIN.MD02.N01_STAT/Device_Info_Data/Project_CRC <-> Device Info Data/Project CRC
//     Standard Inputs/MAIN.MD02.N01_STAT/FBs_FB_ERR @bit 8 <-> StandardInputs/Standard Out Var 13
//     Standard Inputs/MAIN.MD02.N01_STAT/InfoData/AdsAddr/netId <-> InfoData/AdsAddr/netId
//     Standard Inputs/MAIN.MD02.N01_STAT/InfoData/AdsAddr/port <-> InfoData/AdsAddr/port
//     Standard Inputs/MAIN.MD02.N01_STAT/InfoData/State <-> InfoData/State
//     Standard Inputs/MAIN.MD02.N01_STAT/SGs_COM_ERR @bit 1 <-> StandardInputs/Standard Out Var 24
//     Standard Inputs/MAIN.MD02.N01_STAT/SGs_COM_ERR <-> StandardInputs/Standard Out Var 9
//     Standard Inputs/MAIN.MD02.N01_STAT/SGs_FB_ERR <-> StandardInputs/Standard Out Var 10
//     Standard Inputs/MAIN.MD02_N01_I0 <-> StandardInputs/Standard Out Var 40
//     Standard Inputs/MAIN.MD02_N01_I1 <-> StandardInputs/Standard Out Var 41
//     Standard Inputs/MAIN.MD02_N01_I2 <-> StandardInputs/Standard Out Var 42
//     Standard Inputs/MAIN.MD02_N01_I3 <-> StandardInputs/Standard Out Var 43
//     Standard Outputs/MAIN.MD02.N01_CMD/FBs_Restart_Spare <-> StandardOutputs/Standard In Var 23
//     Standard Outputs/MAIN.MD02.N01_CMD/SGs_ERRAck <-> StandardOutputs/Standard In Var 1
//     Standard Outputs/MAIN.MD02.N01_CMD/SGs_ERRAck <-> StandardOutputs/Standard In Var 5
//     Standard Outputs/MAIN.MD02.N01_CMD/SGs_RUNSTOP <-> StandardOutputs/Standard In Var 2
//     Standard Outputs/MAIN.MD02.N01_CMD/SGs_RUNSTOP <-> StandardOutputs/Standard In Var 6
//   SODG11_SSCC610_2403701_PLC/SODG11_SSCC610_2403701_PLC Instance <-> EtherCAT Master (EtherCAT)/MD02.N02 (EP1008-0002)
//     Standard Inputs/MAIN.MD02.N02/I <-> Channel 1/Input
//     Standard Inputs/MAIN.MD02.N02/I @bit 1 <-> Channel 2/Input
//     Standard Inputs/MAIN.MD02.N02/I @bit 2 <-> Channel 3/Input
//     Standard Inputs/MAIN.MD02.N02/I @bit 3 <-> Channel 4/Input
//     Standard Inputs/MAIN.MD02.N02/I @bit 4 <-> Channel 5/Input
//     Standard Inputs/MAIN.MD02.N02/I @bit 5 <-> Channel 6/Input
//     Standard Inputs/MAIN.MD02.N02/I @bit 6 <-> Channel 7/Input
//     Standard Inputs/MAIN.MD02.N02/I @bit 7 <-> Channel 8/Input
//     Standard Inputs/MAIN.MD02.N02/InfoData/State <-> InfoData/State
//   SODG11_SSCC610_2403701_PLC/SODG11_SSCC610_2403701_PLC Instance <-> EtherCAT Master (EtherCAT)/MD02.N03 (EP2624-0002)
//     Standard Inputs/MAIN.MD02.N03_STAT/InfoData/State <-> InfoData/State
//     Standard Outputs/MAIN.MD02.N03/Q <-> Channel 1/Output
//     Standard Outputs/MAIN.MD02.N03/Q @bit 1 <-> Channel 2/Output
//     Standard Outputs/MAIN.MD02.N03/Q @bit 2 <-> Channel 3/Output
//     Standard Outputs/MAIN.MD02.N03/Q @bit 3 <-> Channel 4/Output
//   SODG11_SSCC610_2403701_PLC/SODG11_SSCC610_2403701_PLC Instance <-> EtherCAT Master (EtherCAT)/R1.RT02 (EL6695-1001)
//     Standard Inputs/MAIN.R1.In_From_HW/BYTE_[10] <-> Module 3 (Default IO)/Std. In (64 Bytes)/Input DWORD 2 @bit 8
//     Standard Inputs/MAIN.R1.In_From_HW/BYTE_[11] <-> Module 3 (Default IO)/Std. In (64 Bytes)/Input DWORD 2 @bit 16
//     Standard Inputs/MAIN.R1.In_From_HW/BYTE_[12] <-> Module 3 (Default IO)/Std. In (64 Bytes)/Input DWORD 2 @bit 24
//     Standard Inputs/MAIN.R1.In_From_HW/BYTE_[14] <-> Module 3 (Default IO)/Std. In (64 Bytes)/Input DWORD 3 @bit 8
//     Standard Inputs/MAIN.R1.In_From_HW/BYTE_[15] <-> Module 3 (Default IO)/Std. In (64 Bytes)/Input DWORD 3 @bit 16
//     Standard Inputs/MAIN.R1.In_From_HW/BYTE_[16] <-> Module 3 (Default IO)/Std. In (64 Bytes)/Input DWORD 3 @bit 24
//     Standard Inputs/MAIN.R1.In_From_HW/BYTE_[18] <-> Module 3 (Default IO)/Std. In (64 Bytes)/Input DWORD 4 @bit 8
//     Standard Inputs/MAIN.R1.In_From_HW/BYTE_[19] <-> Module 3 (Default IO)/Std. In (64 Bytes)/Input DWORD 4 @bit 16
//     Standard Inputs/MAIN.R1.In_From_HW/BYTE_[20] <-> Module 3 (Default IO)/Std. In (64 Bytes)/Input DWORD 4 @bit 24
//     Standard Inputs/MAIN.R1.In_From_HW/BYTE_[22] <-> Module 3 (Default IO)/Std. In (64 Bytes)/Input DWORD 5 @bit 8
//     Standard Inputs/MAIN.R1.In_From_HW/BYTE_[23] <-> Module 3 (Default IO)/Std. In (64 Bytes)/Input DWORD 5 @bit 16
//     Standard Inputs/MAIN.R1.In_From_HW/BYTE_[24] <-> Module 3 (Default IO)/Std. In (64 Bytes)/Input DWORD 5 @bit 24
//     Standard Inputs/MAIN.R1.In_From_HW/BYTE_[26] <-> Module 3 (Default IO)/Std. In (64 Bytes)/Input DWORD 6 @bit 8
//     Standard Inputs/MAIN.R1.In_From_HW/BYTE_[27] <-> Module 3 (Default IO)/Std. In (64 Bytes)/Input DWORD 6 @bit 16
//     Standard Inputs/MAIN.R1.In_From_HW/BYTE_[28] <-> Module 3 (Default IO)/Std. In (64 Bytes)/Input DWORD 6 @bit 24
//     Standard Inputs/MAIN.R1.In_From_HW/BYTE_[2] <-> Module 3 (Default IO)/Std. In (64 Bytes)/Input DWORD 0 @bit 8
//     Standard Inputs/MAIN.R1.In_From_HW/BYTE_[30] <-> Module 3 (Default IO)/Std. In (64 Bytes)/Input DWORD 7 @bit 8
//     Standard Inputs/MAIN.R1.In_From_HW/BYTE_[31] <-> Module 3 (Default IO)/Std. In (64 Bytes)/Input DWORD 7 @bit 16
//     Standard Inputs/MAIN.R1.In_From_HW/BYTE_[32] <-> Module 3 (Default IO)/Std. In (64 Bytes)/Input DWORD 7 @bit 24
//     Standard Inputs/MAIN.R1.In_From_HW/BYTE_[34] <-> Module 3 (Default IO)/Std. In (64 Bytes)/Input DWORD 8 @bit 8
//     Standard Inputs/MAIN.R1.In_From_HW/BYTE_[35] <-> Module 3 (Default IO)/Std. In (64 Bytes)/Input DWORD 8 @bit 16
//     Standard Inputs/MAIN.R1.In_From_HW/BYTE_[36] <-> Module 3 (Default IO)/Std. In (64 Bytes)/Input DWORD 8 @bit 24
//     Standard Inputs/MAIN.R1.In_From_HW/BYTE_[38] <-> Module 3 (Default IO)/Std. In (64 Bytes)/Input DWORD 9 @bit 8
//     Standard Inputs/MAIN.R1.In_From_HW/BYTE_[39] <-> Module 3 (Default IO)/Std. In (64 Bytes)/Input DWORD 9 @bit 16
//     Standard Inputs/MAIN.R1.In_From_HW/BYTE_[3] <-> Module 3 (Default IO)/Std. In (64 Bytes)/Input DWORD 0 @bit 16
//     Standard Inputs/MAIN.R1.In_From_HW/BYTE_[40] <-> Module 3 (Default IO)/Std. In (64 Bytes)/Input DWORD 9 @bit 24
//     Standard Inputs/MAIN.R1.In_From_HW/BYTE_[42] <-> Module 3 (Default IO)/Std. In (64 Bytes)/Input DWORD 10 @bit 8
//     Standard Inputs/MAIN.R1.In_From_HW/BYTE_[43] <-> Module 3 (Default IO)/Std. In (64 Bytes)/Input DWORD 10 @bit 16
//     Standard Inputs/MAIN.R1.In_From_HW/BYTE_[44] <-> Module 3 (Default IO)/Std. In (64 Bytes)/Input DWORD 10 @bit 24
//     Standard Inputs/MAIN.R1.In_From_HW/BYTE_[46] <-> Module 3 (Default IO)/Std. In (64 Bytes)/Input DWORD 11 @bit 8
//     Standard Inputs/MAIN.R1.In_From_HW/BYTE_[47] <-> Module 3 (Default IO)/Std. In (64 Bytes)/Input DWORD 11 @bit 16
//     Standard Inputs/MAIN.R1.In_From_HW/BYTE_[48] <-> Module 3 (Default IO)/Std. In (64 Bytes)/Input DWORD 11 @bit 24
//     Standard Inputs/MAIN.R1.In_From_HW/BYTE_[4] <-> Module 3 (Default IO)/Std. In (64 Bytes)/Input DWORD 0 @bit 24
//     Standard Inputs/MAIN.R1.In_From_HW/BYTE_[50] <-> Module 3 (Default IO)/Std. In (64 Bytes)/Input DWORD 12 @bit 8
//     Standard Inputs/MAIN.R1.In_From_HW/BYTE_[51] <-> Module 3 (Default IO)/Std. In (64 Bytes)/Input DWORD 12 @bit 16
//     Standard Inputs/MAIN.R1.In_From_HW/BYTE_[52] <-> Module 3 (Default IO)/Std. In (64 Bytes)/Input DWORD 12 @bit 24
//     Standard Inputs/MAIN.R1.In_From_HW/BYTE_[54] <-> Module 3 (Default IO)/Std. In (64 Bytes)/Input DWORD 13 @bit 8
//     Standard Inputs/MAIN.R1.In_From_HW/BYTE_[55] <-> Module 3 (Default IO)/Std. In (64 Bytes)/Input DWORD 13 @bit 16
//     Standard Inputs/MAIN.R1.In_From_HW/BYTE_[56] <-> Module 3 (Default IO)/Std. In (64 Bytes)/Input DWORD 13 @bit 24
//     Standard Inputs/MAIN.R1.In_From_HW/BYTE_[58] <-> Module 3 (Default IO)/Std. In (64 Bytes)/Input DWORD 14 @bit 8
//     Standard Inputs/MAIN.R1.In_From_HW/BYTE_[59] <-> Module 3 (Default IO)/Std. In (64 Bytes)/Input DWORD 14 @bit 16
//     Standard Inputs/MAIN.R1.In_From_HW/BYTE_[60] <-> Module 3 (Default IO)/Std. In (64 Bytes)/Input DWORD 14 @bit 24
//     Standard Inputs/MAIN.R1.In_From_HW/BYTE_[62] <-> Module 3 (Default IO)/Std. In (64 Bytes)/Input DWORD 15 @bit 8
//     Standard Inputs/MAIN.R1.In_From_HW/BYTE_[63] <-> Module 3 (Default IO)/Std. In (64 Bytes)/Input DWORD 15 @bit 16
//     Standard Inputs/MAIN.R1.In_From_HW/BYTE_[64] <-> Module 3 (Default IO)/Std. In (64 Bytes)/Input DWORD 15 @bit 24
//     Standard Inputs/MAIN.R1.In_From_HW/BYTE_[6] <-> Module 3 (Default IO)/Std. In (64 Bytes)/Input DWORD 1 @bit 8
//     Standard Inputs/MAIN.R1.In_From_HW/BYTE_[7] <-> Module 3 (Default IO)/Std. In (64 Bytes)/Input DWORD 1 @bit 16
//     Standard Inputs/MAIN.R1.In_From_HW/BYTE_[8] <-> Module 3 (Default IO)/Std. In (64 Bytes)/Input DWORD 1 @bit 24
//     Standard Inputs/MAIN.R1.In_From_HW/BYTE_[{1..61 step 4}] <-> Module 3 (Default IO)/Std. In (64 Bytes)/Input DWORD {0..15}  (16 links)
//     Standard Inputs/MAIN.R1.RT02/External_device_not_connected <-> Module 1 (Sync Inputs)/Compact/External device not connected
//     Standard Inputs/MAIN.R1.RT02/FSOE_Inputs_ConnID <-> Module 2 (Safety Data (8 Byte))/Inputs/FSOE/FSOE ConnID
//     Standard Inputs/MAIN.R1.RT02/FSOE_Inputs_Data_0 <-> Module 2 (Safety Data (8 Byte))/Inputs/FSOE/FSOE Data_0
//     Standard Inputs/MAIN.R1.RT02/FSOE_Inputs_Data_1 <-> Module 2 (Safety Data (8 Byte))/Inputs/FSOE/FSOE Data_1
//     Standard Inputs/MAIN.R1.RT02/FSOE_Inputs_Data_2 <-> Module 2 (Safety Data (8 Byte))/Inputs/FSOE/FSOE Data_2
//     Standard Inputs/MAIN.R1.RT02/FSOE_Inputs_Data_3 <-> Module 2 (Safety Data (8 Byte))/Inputs/FSOE/FSOE Data_3
//     Standard Inputs/MAIN.R1.RT02/InfoData/AdsAddr/netId <-> InfoData/AdsAddr/netId
//     Standard Inputs/MAIN.R1.RT02/InfoData/AdsAddr/port <-> InfoData/AdsAddr/port
//     Standard Inputs/MAIN.R1.RT02/InfoData/State <-> InfoData/State
//     Standard Inputs/MAIN.R1.RT02/TxPDO_State <-> Module 1 (Sync Inputs)/Compact/TxPDO state
//     Standard Inputs/MAIN.R1.RT02/TxPDO_Toogle <-> Module 1 (Sync Inputs)/Compact/TxPDO toggle
//     Standard Outputs/MAIN.R1.Out_To_HW/Byte_[10] <-> Module 3 (Default IO)/Std. Out (64 Bytes)/Output DWORD 2 @bit 8
//     Standard Outputs/MAIN.R1.Out_To_HW/Byte_[11] <-> Module 3 (Default IO)/Std. Out (64 Bytes)/Output DWORD 2 @bit 16
//     Standard Outputs/MAIN.R1.Out_To_HW/Byte_[12] <-> Module 3 (Default IO)/Std. Out (64 Bytes)/Output DWORD 2 @bit 24
//     Standard Outputs/MAIN.R1.Out_To_HW/Byte_[14] <-> Module 3 (Default IO)/Std. Out (64 Bytes)/Output DWORD 3 @bit 8
//     Standard Outputs/MAIN.R1.Out_To_HW/Byte_[15] <-> Module 3 (Default IO)/Std. Out (64 Bytes)/Output DWORD 3 @bit 16
//     Standard Outputs/MAIN.R1.Out_To_HW/Byte_[16] <-> Module 3 (Default IO)/Std. Out (64 Bytes)/Output DWORD 3 @bit 24
//     Standard Outputs/MAIN.R1.Out_To_HW/Byte_[18] <-> Module 3 (Default IO)/Std. Out (64 Bytes)/Output DWORD 4 @bit 8
//     Standard Outputs/MAIN.R1.Out_To_HW/Byte_[19] <-> Module 3 (Default IO)/Std. Out (64 Bytes)/Output DWORD 4 @bit 16
//     Standard Outputs/MAIN.R1.Out_To_HW/Byte_[20] <-> Module 3 (Default IO)/Std. Out (64 Bytes)/Output DWORD 4 @bit 24
//     Standard Outputs/MAIN.R1.Out_To_HW/Byte_[22] <-> Module 3 (Default IO)/Std. Out (64 Bytes)/Output DWORD 5 @bit 8
//     Standard Outputs/MAIN.R1.Out_To_HW/Byte_[23] <-> Module 3 (Default IO)/Std. Out (64 Bytes)/Output DWORD 5 @bit 16
//     Standard Outputs/MAIN.R1.Out_To_HW/Byte_[24] <-> Module 3 (Default IO)/Std. Out (64 Bytes)/Output DWORD 5 @bit 24
//     Standard Outputs/MAIN.R1.Out_To_HW/Byte_[26] <-> Module 3 (Default IO)/Std. Out (64 Bytes)/Output DWORD 6 @bit 8
//     Standard Outputs/MAIN.R1.Out_To_HW/Byte_[27] <-> Module 3 (Default IO)/Std. Out (64 Bytes)/Output DWORD 6 @bit 16
//     Standard Outputs/MAIN.R1.Out_To_HW/Byte_[28] <-> Module 3 (Default IO)/Std. Out (64 Bytes)/Output DWORD 6 @bit 24
//     Standard Outputs/MAIN.R1.Out_To_HW/Byte_[2] <-> Module 3 (Default IO)/Std. Out (64 Bytes)/Output DWORD 0 @bit 8
//     Standard Outputs/MAIN.R1.Out_To_HW/Byte_[30] <-> Module 3 (Default IO)/Std. Out (64 Bytes)/Output DWORD 7 @bit 8
//     Standard Outputs/MAIN.R1.Out_To_HW/Byte_[31] <-> Module 3 (Default IO)/Std. Out (64 Bytes)/Output DWORD 7 @bit 16
//     Standard Outputs/MAIN.R1.Out_To_HW/Byte_[32] <-> Module 3 (Default IO)/Std. Out (64 Bytes)/Output DWORD 7 @bit 24
//     Standard Outputs/MAIN.R1.Out_To_HW/Byte_[34] <-> Module 3 (Default IO)/Std. Out (64 Bytes)/Output DWORD 8 @bit 8
//     Standard Outputs/MAIN.R1.Out_To_HW/Byte_[35] <-> Module 3 (Default IO)/Std. Out (64 Bytes)/Output DWORD 8 @bit 16
//     Standard Outputs/MAIN.R1.Out_To_HW/Byte_[36] <-> Module 3 (Default IO)/Std. Out (64 Bytes)/Output DWORD 8 @bit 24
//     Standard Outputs/MAIN.R1.Out_To_HW/Byte_[38] <-> Module 3 (Default IO)/Std. Out (64 Bytes)/Output DWORD 9 @bit 8
//     Standard Outputs/MAIN.R1.Out_To_HW/Byte_[39] <-> Module 3 (Default IO)/Std. Out (64 Bytes)/Output DWORD 9 @bit 16
//     Standard Outputs/MAIN.R1.Out_To_HW/Byte_[3] <-> Module 3 (Default IO)/Std. Out (64 Bytes)/Output DWORD 0 @bit 16
//     Standard Outputs/MAIN.R1.Out_To_HW/Byte_[40] <-> Module 3 (Default IO)/Std. Out (64 Bytes)/Output DWORD 9 @bit 24
//     Standard Outputs/MAIN.R1.Out_To_HW/Byte_[42] <-> Module 3 (Default IO)/Std. Out (64 Bytes)/Output DWORD 10 @bit 8
//     Standard Outputs/MAIN.R1.Out_To_HW/Byte_[43] <-> Module 3 (Default IO)/Std. Out (64 Bytes)/Output DWORD 10 @bit 16
//     Standard Outputs/MAIN.R1.Out_To_HW/Byte_[44] <-> Module 3 (Default IO)/Std. Out (64 Bytes)/Output DWORD 10 @bit 24
//     Standard Outputs/MAIN.R1.Out_To_HW/Byte_[46] <-> Module 3 (Default IO)/Std. Out (64 Bytes)/Output DWORD 11 @bit 8
//     Standard Outputs/MAIN.R1.Out_To_HW/Byte_[47] <-> Module 3 (Default IO)/Std. Out (64 Bytes)/Output DWORD 11 @bit 16
//     Standard Outputs/MAIN.R1.Out_To_HW/Byte_[48] <-> Module 3 (Default IO)/Std. Out (64 Bytes)/Output DWORD 11 @bit 24
//     Standard Outputs/MAIN.R1.Out_To_HW/Byte_[4] <-> Module 3 (Default IO)/Std. Out (64 Bytes)/Output DWORD 0 @bit 24
//     Standard Outputs/MAIN.R1.Out_To_HW/Byte_[50] <-> Module 3 (Default IO)/Std. Out (64 Bytes)/Output DWORD 12 @bit 8
//     Standard Outputs/MAIN.R1.Out_To_HW/Byte_[51] <-> Module 3 (Default IO)/Std. Out (64 Bytes)/Output DWORD 12 @bit 16
//     Standard Outputs/MAIN.R1.Out_To_HW/Byte_[52] <-> Module 3 (Default IO)/Std. Out (64 Bytes)/Output DWORD 12 @bit 24
//     Standard Outputs/MAIN.R1.Out_To_HW/Byte_[54] <-> Module 3 (Default IO)/Std. Out (64 Bytes)/Output DWORD 13 @bit 8
//     Standard Outputs/MAIN.R1.Out_To_HW/Byte_[55] <-> Module 3 (Default IO)/Std. Out (64 Bytes)/Output DWORD 13 @bit 16
//     Standard Outputs/MAIN.R1.Out_To_HW/Byte_[56] <-> Module 3 (Default IO)/Std. Out (64 Bytes)/Output DWORD 13 @bit 24
//     Standard Outputs/MAIN.R1.Out_To_HW/Byte_[58] <-> Module 3 (Default IO)/Std. Out (64 Bytes)/Output DWORD 14 @bit 8
//     Standard Outputs/MAIN.R1.Out_To_HW/Byte_[59] <-> Module 3 (Default IO)/Std. Out (64 Bytes)/Output DWORD 14 @bit 16
//     Standard Outputs/MAIN.R1.Out_To_HW/Byte_[60] <-> Module 3 (Default IO)/Std. Out (64 Bytes)/Output DWORD 14 @bit 24
//     Standard Outputs/MAIN.R1.Out_To_HW/Byte_[62] <-> Module 3 (Default IO)/Std. Out (64 Bytes)/Output DWORD 15 @bit 8
//     Standard Outputs/MAIN.R1.Out_To_HW/Byte_[63] <-> Module 3 (Default IO)/Std. Out (64 Bytes)/Output DWORD 15 @bit 16
//     Standard Outputs/MAIN.R1.Out_To_HW/Byte_[64] <-> Module 3 (Default IO)/Std. Out (64 Bytes)/Output DWORD 15 @bit 24
//     Standard Outputs/MAIN.R1.Out_To_HW/Byte_[6] <-> Module 3 (Default IO)/Std. Out (64 Bytes)/Output DWORD 1 @bit 8
//     Standard Outputs/MAIN.R1.Out_To_HW/Byte_[7] <-> Module 3 (Default IO)/Std. Out (64 Bytes)/Output DWORD 1 @bit 16
//     Standard Outputs/MAIN.R1.Out_To_HW/Byte_[8] <-> Module 3 (Default IO)/Std. Out (64 Bytes)/Output DWORD 1 @bit 24
//     Standard Outputs/MAIN.R1.Out_To_HW/Byte_[{1..61 step 4}] <-> Module 3 (Default IO)/Std. Out (64 Bytes)/Output DWORD {0..15}  (16 links)
//   SODG11_SSCC610_2403701_PLC/SODG11_SSCC610_2403701_PLC Instance <-> EtherCAT Master (EtherCAT)/R1.T01 (EK1100)
//     Standard Inputs/MAIN.R1.T01/InfoData/State <-> InfoData/State
//   SODG11_SSCC610_2403701_PLC/SODG11_SSCC610_2403701_PLC Instance <-> EtherCAT Master (EtherCAT)/R1.T01 (EK1100)/R1.T02 (EL6900)
//     Standard Inputs/MAIN.R1.RT02/FSOE_Outputs_Data_0 @bit 1 <-> StandardInputs/Standard Out Var 14
//     Standard Inputs/MAIN.R1.RT02/FSOE_Outputs_Data_0 @bit 2 <-> StandardInputs/Standard Out Var 15
//     Standard Inputs/MAIN.R1.RT02/FSOE_Outputs_Data_2 @bit 1 <-> StandardInputs/Standard Out Var 18
//     Standard Inputs/MAIN.R1.RT02/FSOE_Outputs_Data_2 @bit 2 <-> StandardInputs/Standard Out Var 19
//     Standard Inputs/MAIN.R1.RT02/FSOE_Outputs_Data_2 @bit 3 <-> StandardInputs/Standard Out Var 20
//     Standard Inputs/MAIN.R1.RT02/FSOE_Outputs_Data_2 <-> StandardInputs/Standard Out Var 17
//     Standard Inputs/MAIN.R1.T02_STAT/Device_Info_Data/Project_CRC <-> Device Info Data/Project CRC
//     Standard Inputs/MAIN.R1.T02_STAT/FBs_FB_ERR <-> StandardInputs/Standard Out Var 16
//     Standard Inputs/MAIN.R1.T02_STAT/FBs_FB_ERR @bit 16 <-> StandardInputs/Standard Out Var 21
//     Standard Inputs/MAIN.R1.T02_STAT/FBs_FB_ERR @bit 29 <-> StandardInputs/Standard Out Var 22
//     Standard Inputs/MAIN.R1.T02_STAT/InfoData/AdsAddr/netId <-> InfoData/AdsAddr/netId
//     Standard Inputs/MAIN.R1.T02_STAT/InfoData/AdsAddr/port <-> InfoData/AdsAddr/port
//     Standard Inputs/MAIN.R1.T02_STAT/InfoData/State <-> InfoData/State
//     Standard Inputs/MAIN.R1.T02_STAT/SGs_COM_ERR @bit 1 <-> StandardInputs/Standard Out Var 12
//     Standard Inputs/MAIN.R1.T02_STAT/SGs_COM_ERR <-> StandardInputs/Standard Out Var 9
//     Standard Inputs/MAIN.R1.T02_STAT/SGs_FB_ERR @bit 1 <-> StandardInputs/Standard Out Var 11
//     Standard Inputs/MAIN.R1.T02_STAT/SGs_FB_ERR <-> StandardInputs/Standard Out Var 8
//     Standard Inputs/MAIN.R1.T02_STAT/SGs_OUT_ERR <-> StandardInputs/Standard Out Var 10
//     Standard Inputs/MAIN.R1.T02_STAT/SGs_OUT_ERR @bit 1 <-> StandardInputs/Standard Out Var 13
//     Standard Outputs/MAIN.R1.T02_CMD/FBs_ControlPowerPB <-> StandardOutputs/Standard In Var 7
//     Standard Outputs/MAIN.R1.T02_CMD/SGs_ERRAck <-> StandardOutputs/Standard In Var 4
//     Standard Outputs/MAIN.R1.T02_CMD/SGs_ERRAck <-> StandardOutputs/Standard In Var 6
//     Standard Outputs/MAIN.R1.T02_CMD/SGs_RUNSTOP <-> StandardOutputs/Standard In Var 3
//     Standard Outputs/MAIN.R1.T02_CMD/SGs_RUNSTOP <-> StandardOutputs/Standard In Var 5
//     Standard Outputs/MAIN.Safety_Zone_Test <-> StandardOutputs/Standard In Var 23
//   SODG11_SSCC610_2403701_PLC/SODG11_SSCC610_2403701_PLC Instance <-> EtherCAT Master (EtherCAT)/R1.T01 (EK1100)/R1.T03 (EL1904)
//     Standard Inputs/MAIN.R1.T03/I <-> Module 1 (FSOES)/TxPDO/FSOE/InputChannel1
//     Standard Inputs/MAIN.R1.T03/I @bit 1 <-> Module 1 (FSOES)/TxPDO/FSOE/InputChannel2
//     Standard Inputs/MAIN.R1.T03/I @bit 2 <-> Module 1 (FSOES)/TxPDO/FSOE/InputChannel3
//     Standard Inputs/MAIN.R1.T03/I @bit 3 <-> Module 1 (FSOES)/TxPDO/FSOE/InputChannel4
//     Standard Inputs/MAIN.R1.T03/InfoData/State <-> InfoData/State
//   SODG11_SSCC610_2403701_PLC/SODG11_SSCC610_2403701_PLC Instance <-> EtherCAT Master (EtherCAT)/R1.T01 (EK1100)/R1.T04 (EK1122)
//     Standard Inputs/MAIN.R1.T04/InfoData/State <-> InfoData/State
//   SODG11_SSCC610_2403701_PLC/SODG11_SSCC610_2403701_PLC Instance <-> EtherCAT Master (EtherCAT)/R1.T01 (EK1100)/R1.T04 (EK1122)/R1.Reamer[1].N01 (EP1008-0002)
//     Standard Inputs/MAIN.R1.Reamer[1].N01/I <-> Channel 1/Input
//     Standard Inputs/MAIN.R1.Reamer[1].N01/I @bit 1 <-> Channel 2/Input
//     Standard Inputs/MAIN.R1.Reamer[1].N01/I @bit 2 <-> Channel 3/Input
//     Standard Inputs/MAIN.R1.Reamer[1].N01/I @bit 3 <-> Channel 4/Input
//     Standard Inputs/MAIN.R1.Reamer[1].N01/I @bit 4 <-> Channel 5/Input
//     Standard Inputs/MAIN.R1.Reamer[1].N01/I @bit 5 <-> Channel 6/Input
//     Standard Inputs/MAIN.R1.Reamer[1].N01/I @bit 6 <-> Channel 7/Input
//     Standard Inputs/MAIN.R1.Reamer[1].N01/I @bit 7 <-> Channel 8/Input
//     Standard Inputs/MAIN.R1.Reamer[1].N01/InfoData/State <-> InfoData/State
//     Standard Inputs/MAIN.R1.Reamer[1].N01/Wc_State <-> WcState/WcState
//   SODG11_SSCC610_2403701_PLC/SODG11_SSCC610_2403701_PLC Instance <-> EtherCAT Master (EtherCAT)/R1.T01 (EK1100)/R1.T04 (EK1122)/R1.Reamer[1].N30 (EP2028-0002)
//     Standard Inputs/MAIN.R1.Reamer[1].N30_STAT/InfoData/State <-> InfoData/State
//     Standard Outputs/MAIN.R1.Reamer[1].N30/Q <-> Channel 1/Output
//     Standard Outputs/MAIN.R1.Reamer[1].N30/Q @bit {1..7} <-> Channel {2..8}/Output  (7 links)
//   SODG11_SSCC610_2403701_PLC/SODG11_SSCC610_2403701_PLC Instance <-> EtherCAT Master (EtherCAT)/R10.RT02 (EL6695-1001)
//     Standard Inputs/MAIN.R10.In_From_HW/BYTE_[10] <-> Module 3 (Default IO)/Std. In (64 Bytes)/Input DWORD 2 @bit 8
//     Standard Inputs/MAIN.R10.In_From_HW/BYTE_[11] <-> Module 3 (Default IO)/Std. In (64 Bytes)/Input DWORD 2 @bit 16
//     Standard Inputs/MAIN.R10.In_From_HW/BYTE_[12] <-> Module 3 (Default IO)/Std. In (64 Bytes)/Input DWORD 2 @bit 24
//     Standard Inputs/MAIN.R10.In_From_HW/BYTE_[14] <-> Module 3 (Default IO)/Std. In (64 Bytes)/Input DWORD 3 @bit 8
//     Standard Inputs/MAIN.R10.In_From_HW/BYTE_[15] <-> Module 3 (Default IO)/Std. In (64 Bytes)/Input DWORD 3 @bit 16
//     Standard Inputs/MAIN.R10.In_From_HW/BYTE_[16] <-> Module 3 (Default IO)/Std. In (64 Bytes)/Input DWORD 3 @bit 24
//     Standard Inputs/MAIN.R10.In_From_HW/BYTE_[18] <-> Module 3 (Default IO)/Std. In (64 Bytes)/Input DWORD 4 @bit 8
//     Standard Inputs/MAIN.R10.In_From_HW/BYTE_[19] <-> Module 3 (Default IO)/Std. In (64 Bytes)/Input DWORD 4 @bit 16
//     Standard Inputs/MAIN.R10.In_From_HW/BYTE_[20] <-> Module 3 (Default IO)/Std. In (64 Bytes)/Input DWORD 4 @bit 24
//     Standard Inputs/MAIN.R10.In_From_HW/BYTE_[22] <-> Module 3 (Default IO)/Std. In (64 Bytes)/Input DWORD 5 @bit 8
//     Standard Inputs/MAIN.R10.In_From_HW/BYTE_[23] <-> Module 3 (Default IO)/Std. In (64 Bytes)/Input DWORD 5 @bit 16
//     Standard Inputs/MAIN.R10.In_From_HW/BYTE_[24] <-> Module 3 (Default IO)/Std. In (64 Bytes)/Input DWORD 5 @bit 24
//     Standard Inputs/MAIN.R10.In_From_HW/BYTE_[26] <-> Module 3 (Default IO)/Std. In (64 Bytes)/Input DWORD 6 @bit 8
//     Standard Inputs/MAIN.R10.In_From_HW/BYTE_[27] <-> Module 3 (Default IO)/Std. In (64 Bytes)/Input DWORD 6 @bit 16
//     Standard Inputs/MAIN.R10.In_From_HW/BYTE_[28] <-> Module 3 (Default IO)/Std. In (64 Bytes)/Input DWORD 6 @bit 24
//     Standard Inputs/MAIN.R10.In_From_HW/BYTE_[2] <-> Module 3 (Default IO)/Std. In (64 Bytes)/Input DWORD 0 @bit 8
//     Standard Inputs/MAIN.R10.In_From_HW/BYTE_[30] <-> Module 3 (Default IO)/Std. In (64 Bytes)/Input DWORD 7 @bit 8
//     Standard Inputs/MAIN.R10.In_From_HW/BYTE_[31] <-> Module 3 (Default IO)/Std. In (64 Bytes)/Input DWORD 7 @bit 16
//     Standard Inputs/MAIN.R10.In_From_HW/BYTE_[32] <-> Module 3 (Default IO)/Std. In (64 Bytes)/Input DWORD 7 @bit 24
//     Standard Inputs/MAIN.R10.In_From_HW/BYTE_[34] <-> Module 3 (Default IO)/Std. In (64 Bytes)/Input DWORD 8 @bit 8
//     Standard Inputs/MAIN.R10.In_From_HW/BYTE_[35] <-> Module 3 (Default IO)/Std. In (64 Bytes)/Input DWORD 8 @bit 16
//     Standard Inputs/MAIN.R10.In_From_HW/BYTE_[36] <-> Module 3 (Default IO)/Std. In (64 Bytes)/Input DWORD 8 @bit 24
//     Standard Inputs/MAIN.R10.In_From_HW/BYTE_[38] <-> Module 3 (Default IO)/Std. In (64 Bytes)/Input DWORD 9 @bit 8
//     Standard Inputs/MAIN.R10.In_From_HW/BYTE_[39] <-> Module 3 (Default IO)/Std. In (64 Bytes)/Input DWORD 9 @bit 16
//     Standard Inputs/MAIN.R10.In_From_HW/BYTE_[3] <-> Module 3 (Default IO)/Std. In (64 Bytes)/Input DWORD 0 @bit 16
//     Standard Inputs/MAIN.R10.In_From_HW/BYTE_[40] <-> Module 3 (Default IO)/Std. In (64 Bytes)/Input DWORD 9 @bit 24
//     Standard Inputs/MAIN.R10.In_From_HW/BYTE_[42] <-> Module 3 (Default IO)/Std. In (64 Bytes)/Input DWORD 10 @bit 8
//     Standard Inputs/MAIN.R10.In_From_HW/BYTE_[43] <-> Module 3 (Default IO)/Std. In (64 Bytes)/Input DWORD 10 @bit 16
//     Standard Inputs/MAIN.R10.In_From_HW/BYTE_[44] <-> Module 3 (Default IO)/Std. In (64 Bytes)/Input DWORD 10 @bit 24
//     Standard Inputs/MAIN.R10.In_From_HW/BYTE_[46] <-> Module 3 (Default IO)/Std. In (64 Bytes)/Input DWORD 11 @bit 8
//     Standard Inputs/MAIN.R10.In_From_HW/BYTE_[47] <-> Module 3 (Default IO)/Std. In (64 Bytes)/Input DWORD 11 @bit 16
//     Standard Inputs/MAIN.R10.In_From_HW/BYTE_[48] <-> Module 3 (Default IO)/Std. In (64 Bytes)/Input DWORD 11 @bit 24
//     Standard Inputs/MAIN.R10.In_From_HW/BYTE_[4] <-> Module 3 (Default IO)/Std. In (64 Bytes)/Input DWORD 0 @bit 24
//     Standard Inputs/MAIN.R10.In_From_HW/BYTE_[50] <-> Module 3 (Default IO)/Std. In (64 Bytes)/Input DWORD 12 @bit 8
//     Standard Inputs/MAIN.R10.In_From_HW/BYTE_[51] <-> Module 3 (Default IO)/Std. In (64 Bytes)/Input DWORD 12 @bit 16
//     Standard Inputs/MAIN.R10.In_From_HW/BYTE_[52] <-> Module 3 (Default IO)/Std. In (64 Bytes)/Input DWORD 12 @bit 24
//     Standard Inputs/MAIN.R10.In_From_HW/BYTE_[54] <-> Module 3 (Default IO)/Std. In (64 Bytes)/Input DWORD 13 @bit 8
//     Standard Inputs/MAIN.R10.In_From_HW/BYTE_[55] <-> Module 3 (Default IO)/Std. In (64 Bytes)/Input DWORD 13 @bit 16
//     Standard Inputs/MAIN.R10.In_From_HW/BYTE_[56] <-> Module 3 (Default IO)/Std. In (64 Bytes)/Input DWORD 13 @bit 24
//     Standard Inputs/MAIN.R10.In_From_HW/BYTE_[58] <-> Module 3 (Default IO)/Std. In (64 Bytes)/Input DWORD 14 @bit 8
//     Standard Inputs/MAIN.R10.In_From_HW/BYTE_[59] <-> Module 3 (Default IO)/Std. In (64 Bytes)/Input DWORD 14 @bit 16
//     Standard Inputs/MAIN.R10.In_From_HW/BYTE_[60] <-> Module 3 (Default IO)/Std. In (64 Bytes)/Input DWORD 14 @bit 24
//     Standard Inputs/MAIN.R10.In_From_HW/BYTE_[62] <-> Module 3 (Default IO)/Std. In (64 Bytes)/Input DWORD 15 @bit 8
//     Standard Inputs/MAIN.R10.In_From_HW/BYTE_[63] <-> Module 3 (Default IO)/Std. In (64 Bytes)/Input DWORD 15 @bit 16
//     Standard Inputs/MAIN.R10.In_From_HW/BYTE_[64] <-> Module 3 (Default IO)/Std. In (64 Bytes)/Input DWORD 15 @bit 24
//     Standard Inputs/MAIN.R10.In_From_HW/BYTE_[6] <-> Module 3 (Default IO)/Std. In (64 Bytes)/Input DWORD 1 @bit 8
//     Standard Inputs/MAIN.R10.In_From_HW/BYTE_[7] <-> Module 3 (Default IO)/Std. In (64 Bytes)/Input DWORD 1 @bit 16
//     Standard Inputs/MAIN.R10.In_From_HW/BYTE_[8] <-> Module 3 (Default IO)/Std. In (64 Bytes)/Input DWORD 1 @bit 24
//     Standard Inputs/MAIN.R10.In_From_HW/BYTE_[{1..61 step 4}] <-> Module 3 (Default IO)/Std. In (64 Bytes)/Input DWORD {0..15}  (16 links)
//     Standard Inputs/MAIN.R10.RT02/External_device_not_connected <-> Module 1 (Sync Inputs)/Compact/External device not connected
//     Standard Inputs/MAIN.R10.RT02/FSOE_Inputs_ConnID <-> Module 2 (Safety Data (8 Byte))/Inputs/FSOE/FSOE ConnID
//     Standard Inputs/MAIN.R10.RT02/FSOE_Inputs_Data_0 <-> Module 2 (Safety Data (8 Byte))/Inputs/FSOE/FSOE Data_0
//     Standard Inputs/MAIN.R10.RT02/FSOE_Inputs_Data_1 <-> Module 2 (Safety Data (8 Byte))/Inputs/FSOE/FSOE Data_1
//     Standard Inputs/MAIN.R10.RT02/FSOE_Inputs_Data_2 <-> Module 2 (Safety Data (8 Byte))/Inputs/FSOE/FSOE Data_2
//     Standard Inputs/MAIN.R10.RT02/FSOE_Inputs_Data_3 <-> Module 2 (Safety Data (8 Byte))/Inputs/FSOE/FSOE Data_3
//     Standard Inputs/MAIN.R10.RT02/InfoData/AdsAddr/netId <-> InfoData/AdsAddr/netId
//     Standard Inputs/MAIN.R10.RT02/InfoData/AdsAddr/port <-> InfoData/AdsAddr/port
//     Standard Inputs/MAIN.R10.RT02/InfoData/State <-> InfoData/State
//     Standard Inputs/MAIN.R10.RT02/TxPDO_State <-> Module 1 (Sync Inputs)/Compact/TxPDO state
//     Standard Inputs/MAIN.R10.RT02/TxPDO_Toogle <-> Module 1 (Sync Inputs)/Compact/TxPDO toggle
//     Standard Outputs/MAIN.R10.Out_To_HW/Byte_[10] <-> Module 3 (Default IO)/Std. Out (64 Bytes)/Output DWORD 2 @bit 8
//     Standard Outputs/MAIN.R10.Out_To_HW/Byte_[11] <-> Module 3 (Default IO)/Std. Out (64 Bytes)/Output DWORD 2 @bit 16
//     Standard Outputs/MAIN.R10.Out_To_HW/Byte_[12] <-> Module 3 (Default IO)/Std. Out (64 Bytes)/Output DWORD 2 @bit 24
//     Standard Outputs/MAIN.R10.Out_To_HW/Byte_[14] <-> Module 3 (Default IO)/Std. Out (64 Bytes)/Output DWORD 3 @bit 8
//     Standard Outputs/MAIN.R10.Out_To_HW/Byte_[15] <-> Module 3 (Default IO)/Std. Out (64 Bytes)/Output DWORD 3 @bit 16
//     Standard Outputs/MAIN.R10.Out_To_HW/Byte_[16] <-> Module 3 (Default IO)/Std. Out (64 Bytes)/Output DWORD 3 @bit 24
//     Standard Outputs/MAIN.R10.Out_To_HW/Byte_[18] <-> Module 3 (Default IO)/Std. Out (64 Bytes)/Output DWORD 4 @bit 8
//     Standard Outputs/MAIN.R10.Out_To_HW/Byte_[19] <-> Module 3 (Default IO)/Std. Out (64 Bytes)/Output DWORD 4 @bit 16
//     Standard Outputs/MAIN.R10.Out_To_HW/Byte_[20] <-> Module 3 (Default IO)/Std. Out (64 Bytes)/Output DWORD 4 @bit 24
//     Standard Outputs/MAIN.R10.Out_To_HW/Byte_[22] <-> Module 3 (Default IO)/Std. Out (64 Bytes)/Output DWORD 5 @bit 8
//     Standard Outputs/MAIN.R10.Out_To_HW/Byte_[23] <-> Module 3 (Default IO)/Std. Out (64 Bytes)/Output DWORD 5 @bit 16
//     Standard Outputs/MAIN.R10.Out_To_HW/Byte_[24] <-> Module 3 (Default IO)/Std. Out (64 Bytes)/Output DWORD 5 @bit 24
//     Standard Outputs/MAIN.R10.Out_To_HW/Byte_[26] <-> Module 3 (Default IO)/Std. Out (64 Bytes)/Output DWORD 6 @bit 8
//     Standard Outputs/MAIN.R10.Out_To_HW/Byte_[27] <-> Module 3 (Default IO)/Std. Out (64 Bytes)/Output DWORD 6 @bit 16
//     Standard Outputs/MAIN.R10.Out_To_HW/Byte_[28] <-> Module 3 (Default IO)/Std. Out (64 Bytes)/Output DWORD 6 @bit 24
//     Standard Outputs/MAIN.R10.Out_To_HW/Byte_[2] <-> Module 3 (Default IO)/Std. Out (64 Bytes)/Output DWORD 0 @bit 8
//     Standard Outputs/MAIN.R10.Out_To_HW/Byte_[30] <-> Module 3 (Default IO)/Std. Out (64 Bytes)/Output DWORD 7 @bit 8
//     Standard Outputs/MAIN.R10.Out_To_HW/Byte_[31] <-> Module 3 (Default IO)/Std. Out (64 Bytes)/Output DWORD 7 @bit 16
//     Standard Outputs/MAIN.R10.Out_To_HW/Byte_[32] <-> Module 3 (Default IO)/Std. Out (64 Bytes)/Output DWORD 7 @bit 24
//     Standard Outputs/MAIN.R10.Out_To_HW/Byte_[34] <-> Module 3 (Default IO)/Std. Out (64 Bytes)/Output DWORD 8 @bit 8
//     Standard Outputs/MAIN.R10.Out_To_HW/Byte_[35] <-> Module 3 (Default IO)/Std. Out (64 Bytes)/Output DWORD 8 @bit 16
//     Standard Outputs/MAIN.R10.Out_To_HW/Byte_[36] <-> Module 3 (Default IO)/Std. Out (64 Bytes)/Output DWORD 8 @bit 24
//     Standard Outputs/MAIN.R10.Out_To_HW/Byte_[38] <-> Module 3 (Default IO)/Std. Out (64 Bytes)/Output DWORD 9 @bit 8
//     Standard Outputs/MAIN.R10.Out_To_HW/Byte_[39] <-> Module 3 (Default IO)/Std. Out (64 Bytes)/Output DWORD 9 @bit 16
//     Standard Outputs/MAIN.R10.Out_To_HW/Byte_[3] <-> Module 3 (Default IO)/Std. Out (64 Bytes)/Output DWORD 0 @bit 16
//     Standard Outputs/MAIN.R10.Out_To_HW/Byte_[40] <-> Module 3 (Default IO)/Std. Out (64 Bytes)/Output DWORD 9 @bit 24
//     Standard Outputs/MAIN.R10.Out_To_HW/Byte_[42] <-> Module 3 (Default IO)/Std. Out (64 Bytes)/Output DWORD 10 @bit 8
//     Standard Outputs/MAIN.R10.Out_To_HW/Byte_[43] <-> Module 3 (Default IO)/Std. Out (64 Bytes)/Output DWORD 10 @bit 16
//     Standard Outputs/MAIN.R10.Out_To_HW/Byte_[44] <-> Module 3 (Default IO)/Std. Out (64 Bytes)/Output DWORD 10 @bit 24
//     Standard Outputs/MAIN.R10.Out_To_HW/Byte_[46] <-> Module 3 (Default IO)/Std. Out (64 Bytes)/Output DWORD 11 @bit 8
//     Standard Outputs/MAIN.R10.Out_To_HW/Byte_[47] <-> Module 3 (Default IO)/Std. Out (64 Bytes)/Output DWORD 11 @bit 16
//     Standard Outputs/MAIN.R10.Out_To_HW/Byte_[48] <-> Module 3 (Default IO)/Std. Out (64 Bytes)/Output DWORD 11 @bit 24
//     Standard Outputs/MAIN.R10.Out_To_HW/Byte_[4] <-> Module 3 (Default IO)/Std. Out (64 Bytes)/Output DWORD 0 @bit 24
//     Standard Outputs/MAIN.R10.Out_To_HW/Byte_[50] <-> Module 3 (Default IO)/Std. Out (64 Bytes)/Output DWORD 12 @bit 8
//     Standard Outputs/MAIN.R10.Out_To_HW/Byte_[51] <-> Module 3 (Default IO)/Std. Out (64 Bytes)/Output DWORD 12 @bit 16
//     Standard Outputs/MAIN.R10.Out_To_HW/Byte_[52] <-> Module 3 (Default IO)/Std. Out (64 Bytes)/Output DWORD 12 @bit 24
//     Standard Outputs/MAIN.R10.Out_To_HW/Byte_[54] <-> Module 3 (Default IO)/Std. Out (64 Bytes)/Output DWORD 13 @bit 8
//     Standard Outputs/MAIN.R10.Out_To_HW/Byte_[55] <-> Module 3 (Default IO)/Std. Out (64 Bytes)/Output DWORD 13 @bit 16
//     Standard Outputs/MAIN.R10.Out_To_HW/Byte_[56] <-> Module 3 (Default IO)/Std. Out (64 Bytes)/Output DWORD 13 @bit 24
//     Standard Outputs/MAIN.R10.Out_To_HW/Byte_[58] <-> Module 3 (Default IO)/Std. Out (64 Bytes)/Output DWORD 14 @bit 8
//     Standard Outputs/MAIN.R10.Out_To_HW/Byte_[59] <-> Module 3 (Default IO)/Std. Out (64 Bytes)/Output DWORD 14 @bit 16
//     Standard Outputs/MAIN.R10.Out_To_HW/Byte_[60] <-> Module 3 (Default IO)/Std. Out (64 Bytes)/Output DWORD 14 @bit 24
//     Standard Outputs/MAIN.R10.Out_To_HW/Byte_[62] <-> Module 3 (Default IO)/Std. Out (64 Bytes)/Output DWORD 15 @bit 8
//     Standard Outputs/MAIN.R10.Out_To_HW/Byte_[63] <-> Module 3 (Default IO)/Std. Out (64 Bytes)/Output DWORD 15 @bit 16
//     Standard Outputs/MAIN.R10.Out_To_HW/Byte_[64] <-> Module 3 (Default IO)/Std. Out (64 Bytes)/Output DWORD 15 @bit 24
//     Standard Outputs/MAIN.R10.Out_To_HW/Byte_[6] <-> Module 3 (Default IO)/Std. Out (64 Bytes)/Output DWORD 1 @bit 8
//     Standard Outputs/MAIN.R10.Out_To_HW/Byte_[7] <-> Module 3 (Default IO)/Std. Out (64 Bytes)/Output DWORD 1 @bit 16
//     Standard Outputs/MAIN.R10.Out_To_HW/Byte_[8] <-> Module 3 (Default IO)/Std. Out (64 Bytes)/Output DWORD 1 @bit 24
//     Standard Outputs/MAIN.R10.Out_To_HW/Byte_[{1..61 step 4}] <-> Module 3 (Default IO)/Std. Out (64 Bytes)/Output DWORD {0..15}  (16 links)
//   SODG11_SSCC610_2403701_PLC/SODG11_SSCC610_2403701_PLC Instance <-> EtherCAT Master (EtherCAT)/R10.T01 (EK1100)
//     Standard Inputs/MAIN.R10.T01/InfoData/State <-> InfoData/State
//   SODG11_SSCC610_2403701_PLC/SODG11_SSCC610_2403701_PLC Instance <-> EtherCAT Master (EtherCAT)/R10.T01 (EK1100)/R10.T02 (EL6900)
//     Standard Inputs/MAIN.R10.RT02/FSOE_Outputs_Data_0 @bit 1 <-> StandardInputs/Standard Out Var 14
//     Standard Inputs/MAIN.R10.RT02/FSOE_Outputs_Data_0 @bit 2 <-> StandardInputs/Standard Out Var 15
//     Standard Inputs/MAIN.R10.RT02/FSOE_Outputs_Data_2 @bit 1 <-> StandardInputs/Standard Out Var 18
//     Standard Inputs/MAIN.R10.RT02/FSOE_Outputs_Data_2 <-> StandardInputs/Standard Out Var 17
//     Standard Inputs/MAIN.R10.T02_STAT/Device_Info_Data/Project_CRC <-> Device Info Data/Project CRC
//     Standard Inputs/MAIN.R10.T02_STAT/FBs_FB_ERR <-> StandardInputs/Standard Out Var 16
//     Standard Inputs/MAIN.R10.T02_STAT/FBs_FB_ERR @bit 16 <-> StandardInputs/Standard Out Var 19
//     Standard Inputs/MAIN.R10.T02_STAT/FBs_FB_ERR @bit 29 <-> StandardInputs/Standard Out Var 20
//     Standard Inputs/MAIN.R10.T02_STAT/InfoData/AdsAddr/netId <-> InfoData/AdsAddr/netId
//     Standard Inputs/MAIN.R10.T02_STAT/InfoData/AdsAddr/port <-> InfoData/AdsAddr/port
//     Standard Inputs/MAIN.R10.T02_STAT/InfoData/State <-> InfoData/State
//     Standard Inputs/MAIN.R10.T02_STAT/SGs_COM_ERR @bit 1 <-> StandardInputs/Standard Out Var 12
//     Standard Inputs/MAIN.R10.T02_STAT/SGs_COM_ERR <-> StandardInputs/Standard Out Var 9
//     Standard Inputs/MAIN.R10.T02_STAT/SGs_FB_ERR @bit 1 <-> StandardInputs/Standard Out Var 11
//     Standard Inputs/MAIN.R10.T02_STAT/SGs_FB_ERR <-> StandardInputs/Standard Out Var 8
//     Standard Inputs/MAIN.R10.T02_STAT/SGs_OUT_ERR <-> StandardInputs/Standard Out Var 10
//     Standard Inputs/MAIN.R10.T02_STAT/SGs_OUT_ERR @bit 1 <-> StandardInputs/Standard Out Var 13
//     Standard Outputs/MAIN.R10.T02_CMD/FBs_ControlPowerPB <-> StandardOutputs/Standard In Var 7
//     Standard Outputs/MAIN.R10.T02_CMD/SGs_ERRAck <-> StandardOutputs/Standard In Var 4
//     Standard Outputs/MAIN.R10.T02_CMD/SGs_ERRAck <-> StandardOutputs/Standard In Var 6
//     Standard Outputs/MAIN.R10.T02_CMD/SGs_RUNSTOP <-> StandardOutputs/Standard In Var 3
//     Standard Outputs/MAIN.R10.T02_CMD/SGs_RUNSTOP <-> StandardOutputs/Standard In Var 5
//     Standard Outputs/MAIN.Safety_Zone_Test <-> StandardOutputs/Standard In Var 21
//   SODG11_SSCC610_2403701_PLC/SODG11_SSCC610_2403701_PLC Instance <-> EtherCAT Master (EtherCAT)/R10.T01 (EK1100)/R10.T03 (EL1904)
//     Standard Inputs/MAIN.R10.T03/I <-> Module 1 (FSOES)/TxPDO/FSOE/InputChannel1
//     Standard Inputs/MAIN.R10.T03/I @bit 1 <-> Module 1 (FSOES)/TxPDO/FSOE/InputChannel2
//     Standard Inputs/MAIN.R10.T03/I @bit 2 <-> Module 1 (FSOES)/TxPDO/FSOE/InputChannel3
//     Standard Inputs/MAIN.R10.T03/I @bit 3 <-> Module 1 (FSOES)/TxPDO/FSOE/InputChannel4
//     Standard Inputs/MAIN.R10.T03/InfoData/State <-> InfoData/State
//   SODG11_SSCC610_2403701_PLC/SODG11_SSCC610_2403701_PLC Instance <-> EtherCAT Master (EtherCAT)/R10.T01 (EK1100)/R10.T04 (EK1122)
//     Standard Inputs/MAIN.R10.T04/InfoData/State <-> InfoData/State
//   SODG11_SSCC610_2403701_PLC/SODG11_SSCC610_2403701_PLC Instance <-> EtherCAT Master (EtherCAT)/R11.RT02 (EL6695-1001)
//     Standard Inputs/MAIN.R11.In_From_HW/BYTE_[10] <-> Module 3 (Default IO)/Std. In (64 Bytes)/Input DWORD 2 @bit 8
//     Standard Inputs/MAIN.R11.In_From_HW/BYTE_[11] <-> Module 3 (Default IO)/Std. In (64 Bytes)/Input DWORD 2 @bit 16
//     Standard Inputs/MAIN.R11.In_From_HW/BYTE_[12] <-> Module 3 (Default IO)/Std. In (64 Bytes)/Input DWORD 2 @bit 24
//     Standard Inputs/MAIN.R11.In_From_HW/BYTE_[14] <-> Module 3 (Default IO)/Std. In (64 Bytes)/Input DWORD 3 @bit 8
//     Standard Inputs/MAIN.R11.In_From_HW/BYTE_[15] <-> Module 3 (Default IO)/Std. In (64 Bytes)/Input DWORD 3 @bit 16
//     Standard Inputs/MAIN.R11.In_From_HW/BYTE_[16] <-> Module 3 (Default IO)/Std. In (64 Bytes)/Input DWORD 3 @bit 24
//     Standard Inputs/MAIN.R11.In_From_HW/BYTE_[18] <-> Module 3 (Default IO)/Std. In (64 Bytes)/Input DWORD 4 @bit 8
//     Standard Inputs/MAIN.R11.In_From_HW/BYTE_[19] <-> Module 3 (Default IO)/Std. In (64 Bytes)/Input DWORD 4 @bit 16
//     Standard Inputs/MAIN.R11.In_From_HW/BYTE_[20] <-> Module 3 (Default IO)/Std. In (64 Bytes)/Input DWORD 4 @bit 24
//     Standard Inputs/MAIN.R11.In_From_HW/BYTE_[22] <-> Module 3 (Default IO)/Std. In (64 Bytes)/Input DWORD 5 @bit 8
//     Standard Inputs/MAIN.R11.In_From_HW/BYTE_[23] <-> Module 3 (Default IO)/Std. In (64 Bytes)/Input DWORD 5 @bit 16
//     Standard Inputs/MAIN.R11.In_From_HW/BYTE_[24] <-> Module 3 (Default IO)/Std. In (64 Bytes)/Input DWORD 5 @bit 24
//     Standard Inputs/MAIN.R11.In_From_HW/BYTE_[26] <-> Module 3 (Default IO)/Std. In (64 Bytes)/Input DWORD 6 @bit 8
//     Standard Inputs/MAIN.R11.In_From_HW/BYTE_[27] <-> Module 3 (Default IO)/Std. In (64 Bytes)/Input DWORD 6 @bit 16
//     Standard Inputs/MAIN.R11.In_From_HW/BYTE_[28] <-> Module 3 (Default IO)/Std. In (64 Bytes)/Input DWORD 6 @bit 24
//     Standard Inputs/MAIN.R11.In_From_HW/BYTE_[2] <-> Module 3 (Default IO)/Std. In (64 Bytes)/Input DWORD 0 @bit 8
//     Standard Inputs/MAIN.R11.In_From_HW/BYTE_[30] <-> Module 3 (Default IO)/Std. In (64 Bytes)/Input DWORD 7 @bit 8
//     Standard Inputs/MAIN.R11.In_From_HW/BYTE_[31] <-> Module 3 (Default IO)/Std. In (64 Bytes)/Input DWORD 7 @bit 16
//     Standard Inputs/MAIN.R11.In_From_HW/BYTE_[32] <-> Module 3 (Default IO)/Std. In (64 Bytes)/Input DWORD 7 @bit 24
//     Standard Inputs/MAIN.R11.In_From_HW/BYTE_[34] <-> Module 3 (Default IO)/Std. In (64 Bytes)/Input DWORD 8 @bit 8
//     Standard Inputs/MAIN.R11.In_From_HW/BYTE_[35] <-> Module 3 (Default IO)/Std. In (64 Bytes)/Input DWORD 8 @bit 16
//     Standard Inputs/MAIN.R11.In_From_HW/BYTE_[36] <-> Module 3 (Default IO)/Std. In (64 Bytes)/Input DWORD 8 @bit 24
//     Standard Inputs/MAIN.R11.In_From_HW/BYTE_[38] <-> Module 3 (Default IO)/Std. In (64 Bytes)/Input DWORD 9 @bit 8
//     Standard Inputs/MAIN.R11.In_From_HW/BYTE_[39] <-> Module 3 (Default IO)/Std. In (64 Bytes)/Input DWORD 9 @bit 16
//     Standard Inputs/MAIN.R11.In_From_HW/BYTE_[3] <-> Module 3 (Default IO)/Std. In (64 Bytes)/Input DWORD 0 @bit 16
//     Standard Inputs/MAIN.R11.In_From_HW/BYTE_[40] <-> Module 3 (Default IO)/Std. In (64 Bytes)/Input DWORD 9 @bit 24
//     Standard Inputs/MAIN.R11.In_From_HW/BYTE_[42] <-> Module 3 (Default IO)/Std. In (64 Bytes)/Input DWORD 10 @bit 8
//     Standard Inputs/MAIN.R11.In_From_HW/BYTE_[43] <-> Module 3 (Default IO)/Std. In (64 Bytes)/Input DWORD 10 @bit 16
//     Standard Inputs/MAIN.R11.In_From_HW/BYTE_[44] <-> Module 3 (Default IO)/Std. In (64 Bytes)/Input DWORD 10 @bit 24
//     Standard Inputs/MAIN.R11.In_From_HW/BYTE_[46] <-> Module 3 (Default IO)/Std. In (64 Bytes)/Input DWORD 11 @bit 8
//     Standard Inputs/MAIN.R11.In_From_HW/BYTE_[47] <-> Module 3 (Default IO)/Std. In (64 Bytes)/Input DWORD 11 @bit 16
//     Standard Inputs/MAIN.R11.In_From_HW/BYTE_[48] <-> Module 3 (Default IO)/Std. In (64 Bytes)/Input DWORD 11 @bit 24
//     Standard Inputs/MAIN.R11.In_From_HW/BYTE_[4] <-> Module 3 (Default IO)/Std. In (64 Bytes)/Input DWORD 0 @bit 24
//     Standard Inputs/MAIN.R11.In_From_HW/BYTE_[50] <-> Module 3 (Default IO)/Std. In (64 Bytes)/Input DWORD 12 @bit 8
//     Standard Inputs/MAIN.R11.In_From_HW/BYTE_[51] <-> Module 3 (Default IO)/Std. In (64 Bytes)/Input DWORD 12 @bit 16
//     Standard Inputs/MAIN.R11.In_From_HW/BYTE_[52] <-> Module 3 (Default IO)/Std. In (64 Bytes)/Input DWORD 12 @bit 24
//     Standard Inputs/MAIN.R11.In_From_HW/BYTE_[54] <-> Module 3 (Default IO)/Std. In (64 Bytes)/Input DWORD 13 @bit 8
//     Standard Inputs/MAIN.R11.In_From_HW/BYTE_[55] <-> Module 3 (Default IO)/Std. In (64 Bytes)/Input DWORD 13 @bit 16
//     Standard Inputs/MAIN.R11.In_From_HW/BYTE_[56] <-> Module 3 (Default IO)/Std. In (64 Bytes)/Input DWORD 13 @bit 24
//     Standard Inputs/MAIN.R11.In_From_HW/BYTE_[58] <-> Module 3 (Default IO)/Std. In (64 Bytes)/Input DWORD 14 @bit 8
//     Standard Inputs/MAIN.R11.In_From_HW/BYTE_[59] <-> Module 3 (Default IO)/Std. In (64 Bytes)/Input DWORD 14 @bit 16
//     Standard Inputs/MAIN.R11.In_From_HW/BYTE_[60] <-> Module 3 (Default IO)/Std. In (64 Bytes)/Input DWORD 14 @bit 24
//     Standard Inputs/MAIN.R11.In_From_HW/BYTE_[62] <-> Module 3 (Default IO)/Std. In (64 Bytes)/Input DWORD 15 @bit 8
//     Standard Inputs/MAIN.R11.In_From_HW/BYTE_[63] <-> Module 3 (Default IO)/Std. In (64 Bytes)/Input DWORD 15 @bit 16
//     Standard Inputs/MAIN.R11.In_From_HW/BYTE_[64] <-> Module 3 (Default IO)/Std. In (64 Bytes)/Input DWORD 15 @bit 24
//     Standard Inputs/MAIN.R11.In_From_HW/BYTE_[6] <-> Module 3 (Default IO)/Std. In (64 Bytes)/Input DWORD 1 @bit 8
//     Standard Inputs/MAIN.R11.In_From_HW/BYTE_[7] <-> Module 3 (Default IO)/Std. In (64 Bytes)/Input DWORD 1 @bit 16
//     Standard Inputs/MAIN.R11.In_From_HW/BYTE_[8] <-> Module 3 (Default IO)/Std. In (64 Bytes)/Input DWORD 1 @bit 24
//     Standard Inputs/MAIN.R11.In_From_HW/BYTE_[{1..61 step 4}] <-> Module 3 (Default IO)/Std. In (64 Bytes)/Input DWORD {0..15}  (16 links)
//     Standard Inputs/MAIN.R11.RT02/External_device_not_connected <-> Module 1 (Sync Inputs)/Compact/External device not connected
//     Standard Inputs/MAIN.R11.RT02/FSOE_Inputs_ConnID <-> Module 2 (Safety Data (8 Byte))/Inputs/FSOE/FSOE ConnID
//     Standard Inputs/MAIN.R11.RT02/FSOE_Inputs_Data_0 <-> Module 2 (Safety Data (8 Byte))/Inputs/FSOE/FSOE Data_0
//     Standard Inputs/MAIN.R11.RT02/FSOE_Inputs_Data_1 <-> Module 2 (Safety Data (8 Byte))/Inputs/FSOE/FSOE Data_1
//     Standard Inputs/MAIN.R11.RT02/FSOE_Inputs_Data_2 <-> Module 2 (Safety Data (8 Byte))/Inputs/FSOE/FSOE Data_2
//     Standard Inputs/MAIN.R11.RT02/FSOE_Inputs_Data_3 <-> Module 2 (Safety Data (8 Byte))/Inputs/FSOE/FSOE Data_3
//     Standard Inputs/MAIN.R11.RT02/InfoData/AdsAddr/netId <-> InfoData/AdsAddr/netId
//     Standard Inputs/MAIN.R11.RT02/InfoData/AdsAddr/port <-> InfoData/AdsAddr/port
//     Standard Inputs/MAIN.R11.RT02/InfoData/State <-> InfoData/State
//     Standard Inputs/MAIN.R11.RT02/TxPDO_State <-> Module 1 (Sync Inputs)/Compact/TxPDO state
//     Standard Inputs/MAIN.R11.RT02/TxPDO_Toogle <-> Module 1 (Sync Inputs)/Compact/TxPDO toggle
//     Standard Outputs/MAIN.R11.Out_To_HW/Byte_[10] <-> Module 3 (Default IO)/Std. Out (64 Bytes)/Output DWORD 2 @bit 8
//     Standard Outputs/MAIN.R11.Out_To_HW/Byte_[11] <-> Module 3 (Default IO)/Std. Out (64 Bytes)/Output DWORD 2 @bit 16
//     Standard Outputs/MAIN.R11.Out_To_HW/Byte_[12] <-> Module 3 (Default IO)/Std. Out (64 Bytes)/Output DWORD 2 @bit 24
//     Standard Outputs/MAIN.R11.Out_To_HW/Byte_[14] <-> Module 3 (Default IO)/Std. Out (64 Bytes)/Output DWORD 3 @bit 8
//     Standard Outputs/MAIN.R11.Out_To_HW/Byte_[15] <-> Module 3 (Default IO)/Std. Out (64 Bytes)/Output DWORD 3 @bit 16
//     Standard Outputs/MAIN.R11.Out_To_HW/Byte_[16] <-> Module 3 (Default IO)/Std. Out (64 Bytes)/Output DWORD 3 @bit 24
//     Standard Outputs/MAIN.R11.Out_To_HW/Byte_[18] <-> Module 3 (Default IO)/Std. Out (64 Bytes)/Output DWORD 4 @bit 8
//     Standard Outputs/MAIN.R11.Out_To_HW/Byte_[19] <-> Module 3 (Default IO)/Std. Out (64 Bytes)/Output DWORD 4 @bit 16
//     Standard Outputs/MAIN.R11.Out_To_HW/Byte_[20] <-> Module 3 (Default IO)/Std. Out (64 Bytes)/Output DWORD 4 @bit 24
//     Standard Outputs/MAIN.R11.Out_To_HW/Byte_[22] <-> Module 3 (Default IO)/Std. Out (64 Bytes)/Output DWORD 5 @bit 8
//     Standard Outputs/MAIN.R11.Out_To_HW/Byte_[23] <-> Module 3 (Default IO)/Std. Out (64 Bytes)/Output DWORD 5 @bit 16
//     Standard Outputs/MAIN.R11.Out_To_HW/Byte_[24] <-> Module 3 (Default IO)/Std. Out (64 Bytes)/Output DWORD 5 @bit 24
//     Standard Outputs/MAIN.R11.Out_To_HW/Byte_[26] <-> Module 3 (Default IO)/Std. Out (64 Bytes)/Output DWORD 6 @bit 8
//     Standard Outputs/MAIN.R11.Out_To_HW/Byte_[27] <-> Module 3 (Default IO)/Std. Out (64 Bytes)/Output DWORD 6 @bit 16
//     Standard Outputs/MAIN.R11.Out_To_HW/Byte_[28] <-> Module 3 (Default IO)/Std. Out (64 Bytes)/Output DWORD 6 @bit 24
//     Standard Outputs/MAIN.R11.Out_To_HW/Byte_[2] <-> Module 3 (Default IO)/Std. Out (64 Bytes)/Output DWORD 0 @bit 8
//     Standard Outputs/MAIN.R11.Out_To_HW/Byte_[30] <-> Module 3 (Default IO)/Std. Out (64 Bytes)/Output DWORD 7 @bit 8
//     Standard Outputs/MAIN.R11.Out_To_HW/Byte_[31] <-> Module 3 (Default IO)/Std. Out (64 Bytes)/Output DWORD 7 @bit 16
//     Standard Outputs/MAIN.R11.Out_To_HW/Byte_[32] <-> Module 3 (Default IO)/Std. Out (64 Bytes)/Output DWORD 7 @bit 24
//     Standard Outputs/MAIN.R11.Out_To_HW/Byte_[34] <-> Module 3 (Default IO)/Std. Out (64 Bytes)/Output DWORD 8 @bit 8
//     Standard Outputs/MAIN.R11.Out_To_HW/Byte_[35] <-> Module 3 (Default IO)/Std. Out (64 Bytes)/Output DWORD 8 @bit 16
//     Standard Outputs/MAIN.R11.Out_To_HW/Byte_[36] <-> Module 3 (Default IO)/Std. Out (64 Bytes)/Output DWORD 8 @bit 24
//     Standard Outputs/MAIN.R11.Out_To_HW/Byte_[38] <-> Module 3 (Default IO)/Std. Out (64 Bytes)/Output DWORD 9 @bit 8
//     Standard Outputs/MAIN.R11.Out_To_HW/Byte_[39] <-> Module 3 (Default IO)/Std. Out (64 Bytes)/Output DWORD 9 @bit 16
//     Standard Outputs/MAIN.R11.Out_To_HW/Byte_[3] <-> Module 3 (Default IO)/Std. Out (64 Bytes)/Output DWORD 0 @bit 16
//     Standard Outputs/MAIN.R11.Out_To_HW/Byte_[40] <-> Module 3 (Default IO)/Std. Out (64 Bytes)/Output DWORD 9 @bit 24
//     Standard Outputs/MAIN.R11.Out_To_HW/Byte_[42] <-> Module 3 (Default IO)/Std. Out (64 Bytes)/Output DWORD 10 @bit 8
//     Standard Outputs/MAIN.R11.Out_To_HW/Byte_[43] <-> Module 3 (Default IO)/Std. Out (64 Bytes)/Output DWORD 10 @bit 16
//     Standard Outputs/MAIN.R11.Out_To_HW/Byte_[44] <-> Module 3 (Default IO)/Std. Out (64 Bytes)/Output DWORD 10 @bit 24
//     Standard Outputs/MAIN.R11.Out_To_HW/Byte_[46] <-> Module 3 (Default IO)/Std. Out (64 Bytes)/Output DWORD 11 @bit 8
//     Standard Outputs/MAIN.R11.Out_To_HW/Byte_[47] <-> Module 3 (Default IO)/Std. Out (64 Bytes)/Output DWORD 11 @bit 16
//     Standard Outputs/MAIN.R11.Out_To_HW/Byte_[48] <-> Module 3 (Default IO)/Std. Out (64 Bytes)/Output DWORD 11 @bit 24
//     Standard Outputs/MAIN.R11.Out_To_HW/Byte_[4] <-> Module 3 (Default IO)/Std. Out (64 Bytes)/Output DWORD 0 @bit 24
//     Standard Outputs/MAIN.R11.Out_To_HW/Byte_[50] <-> Module 3 (Default IO)/Std. Out (64 Bytes)/Output DWORD 12 @bit 8
//     Standard Outputs/MAIN.R11.Out_To_HW/Byte_[51] <-> Module 3 (Default IO)/Std. Out (64 Bytes)/Output DWORD 12 @bit 16
//     Standard Outputs/MAIN.R11.Out_To_HW/Byte_[52] <-> Module 3 (Default IO)/Std. Out (64 Bytes)/Output DWORD 12 @bit 24
//     Standard Outputs/MAIN.R11.Out_To_HW/Byte_[54] <-> Module 3 (Default IO)/Std. Out (64 Bytes)/Output DWORD 13 @bit 8
//     Standard Outputs/MAIN.R11.Out_To_HW/Byte_[55] <-> Module 3 (Default IO)/Std. Out (64 Bytes)/Output DWORD 13 @bit 16
//     Standard Outputs/MAIN.R11.Out_To_HW/Byte_[56] <-> Module 3 (Default IO)/Std. Out (64 Bytes)/Output DWORD 13 @bit 24
//     Standard Outputs/MAIN.R11.Out_To_HW/Byte_[58] <-> Module 3 (Default IO)/Std. Out (64 Bytes)/Output DWORD 14 @bit 8
//     Standard Outputs/MAIN.R11.Out_To_HW/Byte_[59] <-> Module 3 (Default IO)/Std. Out (64 Bytes)/Output DWORD 14 @bit 16
//     Standard Outputs/MAIN.R11.Out_To_HW/Byte_[60] <-> Module 3 (Default IO)/Std. Out (64 Bytes)/Output DWORD 14 @bit 24
//     Standard Outputs/MAIN.R11.Out_To_HW/Byte_[62] <-> Module 3 (Default IO)/Std. Out (64 Bytes)/Output DWORD 15 @bit 8
//     Standard Outputs/MAIN.R11.Out_To_HW/Byte_[63] <-> Module 3 (Default IO)/Std. Out (64 Bytes)/Output DWORD 15 @bit 16
//     Standard Outputs/MAIN.R11.Out_To_HW/Byte_[64] <-> Module 3 (Default IO)/Std. Out (64 Bytes)/Output DWORD 15 @bit 24
//     Standard Outputs/MAIN.R11.Out_To_HW/Byte_[6] <-> Module 3 (Default IO)/Std. Out (64 Bytes)/Output DWORD 1 @bit 8
//     Standard Outputs/MAIN.R11.Out_To_HW/Byte_[7] <-> Module 3 (Default IO)/Std. Out (64 Bytes)/Output DWORD 1 @bit 16
//     Standard Outputs/MAIN.R11.Out_To_HW/Byte_[8] <-> Module 3 (Default IO)/Std. Out (64 Bytes)/Output DWORD 1 @bit 24
//     Standard Outputs/MAIN.R11.Out_To_HW/Byte_[{1..61 step 4}] <-> Module 3 (Default IO)/Std. Out (64 Bytes)/Output DWORD {0..15}  (16 links)
//   SODG11_SSCC610_2403701_PLC/SODG11_SSCC610_2403701_PLC Instance <-> EtherCAT Master (EtherCAT)/R11.T01 (EK1100)
//     Standard Inputs/MAIN.R11.T01/InfoData/State <-> InfoData/State
//   SODG11_SSCC610_2403701_PLC/SODG11_SSCC610_2403701_PLC Instance <-> EtherCAT Master (EtherCAT)/R11.T01 (EK1100)/R11.T02 (EL6900)
//     Standard Inputs/MAIN.R11.RT02/FSOE_Outputs_Data_0 @bit 1 <-> StandardInputs/Standard Out Var 14
//     Standard Inputs/MAIN.R11.RT02/FSOE_Outputs_Data_0 @bit 2 <-> StandardInputs/Standard Out Var 15
//     Standard Inputs/MAIN.R11.RT02/FSOE_Outputs_Data_2 @bit 1 <-> StandardInputs/Standard Out Var 18
//     Standard Inputs/MAIN.R11.RT02/FSOE_Outputs_Data_2 <-> StandardInputs/Standard Out Var 17
//     Standard Inputs/MAIN.R11.T02_STAT/Device_Info_Data/Project_CRC <-> Device Info Data/Project CRC
//     Standard Inputs/MAIN.R11.T02_STAT/FBs_FB_ERR <-> StandardInputs/Standard Out Var 16
//     Standard Inputs/MAIN.R11.T02_STAT/FBs_FB_ERR @bit 16 <-> StandardInputs/Standard Out Var 19
//     Standard Inputs/MAIN.R11.T02_STAT/FBs_FB_ERR @bit 29 <-> StandardInputs/Standard Out Var 20
//     Standard Inputs/MAIN.R11.T02_STAT/InfoData/AdsAddr/netId <-> InfoData/AdsAddr/netId
//     Standard Inputs/MAIN.R11.T02_STAT/InfoData/AdsAddr/port <-> InfoData/AdsAddr/port
//     Standard Inputs/MAIN.R11.T02_STAT/InfoData/State <-> InfoData/State
//     Standard Inputs/MAIN.R11.T02_STAT/SGs_COM_ERR @bit 1 <-> StandardInputs/Standard Out Var 12
//     Standard Inputs/MAIN.R11.T02_STAT/SGs_COM_ERR <-> StandardInputs/Standard Out Var 9
//     Standard Inputs/MAIN.R11.T02_STAT/SGs_FB_ERR @bit 1 <-> StandardInputs/Standard Out Var 11
//     Standard Inputs/MAIN.R11.T02_STAT/SGs_FB_ERR <-> StandardInputs/Standard Out Var 8
//     Standard Inputs/MAIN.R11.T02_STAT/SGs_OUT_ERR <-> StandardInputs/Standard Out Var 10
//     Standard Inputs/MAIN.R11.T02_STAT/SGs_OUT_ERR @bit 1 <-> StandardInputs/Standard Out Var 13
//     Standard Outputs/MAIN.R11.T02_CMD/FBs_ControlPowerPB <-> StandardOutputs/Standard In Var 7
//     Standard Outputs/MAIN.R11.T02_CMD/SGs_ERRAck <-> StandardOutputs/Standard In Var 4
//     Standard Outputs/MAIN.R11.T02_CMD/SGs_ERRAck <-> StandardOutputs/Standard In Var 6
//     Standard Outputs/MAIN.R11.T02_CMD/SGs_RUNSTOP <-> StandardOutputs/Standard In Var 3
//     Standard Outputs/MAIN.R11.T02_CMD/SGs_RUNSTOP <-> StandardOutputs/Standard In Var 5
//     Standard Outputs/MAIN.Safety_Zone_Test <-> StandardOutputs/Standard In Var 21
//   SODG11_SSCC610_2403701_PLC/SODG11_SSCC610_2403701_PLC Instance <-> EtherCAT Master (EtherCAT)/R11.T01 (EK1100)/R11.T03 (EL1904)
//     Standard Inputs/MAIN.R11.T03/I <-> Module 1 (FSOES)/TxPDO/FSOE/InputChannel1
//     Standard Inputs/MAIN.R11.T03/I @bit 1 <-> Module 1 (FSOES)/TxPDO/FSOE/InputChannel2
//     Standard Inputs/MAIN.R11.T03/I @bit 2 <-> Module 1 (FSOES)/TxPDO/FSOE/InputChannel3
//     Standard Inputs/MAIN.R11.T03/I @bit 3 <-> Module 1 (FSOES)/TxPDO/FSOE/InputChannel4
//     Standard Inputs/MAIN.R11.T03/InfoData/State <-> InfoData/State
//   SODG11_SSCC610_2403701_PLC/SODG11_SSCC610_2403701_PLC Instance <-> EtherCAT Master (EtherCAT)/R11.T01 (EK1100)/R11.T04 (EK1122)
//     Standard Inputs/MAIN.R11.T04/InfoData/State <-> InfoData/State
//   SODG11_SSCC610_2403701_PLC/SODG11_SSCC610_2403701_PLC Instance <-> EtherCAT Master (EtherCAT)/R2.RT02 (EL6695-1001)
//     Standard Inputs/MAIN.R2.In_From_HW/BYTE_[10] <-> Module 3 (Default IO)/Std. In (64 Bytes)/Input DWORD 2 @bit 8
//     Standard Inputs/MAIN.R2.In_From_HW/BYTE_[11] <-> Module 3 (Default IO)/Std. In (64 Bytes)/Input DWORD 2 @bit 16
//     Standard Inputs/MAIN.R2.In_From_HW/BYTE_[12] <-> Module 3 (Default IO)/Std. In (64 Bytes)/Input DWORD 2 @bit 24
//     Standard Inputs/MAIN.R2.In_From_HW/BYTE_[14] <-> Module 3 (Default IO)/Std. In (64 Bytes)/Input DWORD 3 @bit 8
//     Standard Inputs/MAIN.R2.In_From_HW/BYTE_[15] <-> Module 3 (Default IO)/Std. In (64 Bytes)/Input DWORD 3 @bit 16
//     Standard Inputs/MAIN.R2.In_From_HW/BYTE_[16] <-> Module 3 (Default IO)/Std. In (64 Bytes)/Input DWORD 3 @bit 24
//     Standard Inputs/MAIN.R2.In_From_HW/BYTE_[18] <-> Module 3 (Default IO)/Std. In (64 Bytes)/Input DWORD 4 @bit 8
//     Standard Inputs/MAIN.R2.In_From_HW/BYTE_[19] <-> Module 3 (Default IO)/Std. In (64 Bytes)/Input DWORD 4 @bit 16
//     Standard Inputs/MAIN.R2.In_From_HW/BYTE_[20] <-> Module 3 (Default IO)/Std. In (64 Bytes)/Input DWORD 4 @bit 24
//     Standard Inputs/MAIN.R2.In_From_HW/BYTE_[22] <-> Module 3 (Default IO)/Std. In (64 Bytes)/Input DWORD 5 @bit 8
//     Standard Inputs/MAIN.R2.In_From_HW/BYTE_[23] <-> Module 3 (Default IO)/Std. In (64 Bytes)/Input DWORD 5 @bit 16
//     Standard Inputs/MAIN.R2.In_From_HW/BYTE_[24] <-> Module 3 (Default IO)/Std. In (64 Bytes)/Input DWORD 5 @bit 24
//     Standard Inputs/MAIN.R2.In_From_HW/BYTE_[26] <-> Module 3 (Default IO)/Std. In (64 Bytes)/Input DWORD 6 @bit 8
//     Standard Inputs/MAIN.R2.In_From_HW/BYTE_[27] <-> Module 3 (Default IO)/Std. In (64 Bytes)/Input DWORD 6 @bit 16
//     Standard Inputs/MAIN.R2.In_From_HW/BYTE_[28] <-> Module 3 (Default IO)/Std. In (64 Bytes)/Input DWORD 6 @bit 24
//     Standard Inputs/MAIN.R2.In_From_HW/BYTE_[2] <-> Module 3 (Default IO)/Std. In (64 Bytes)/Input DWORD 0 @bit 8
//     Standard Inputs/MAIN.R2.In_From_HW/BYTE_[30] <-> Module 3 (Default IO)/Std. In (64 Bytes)/Input DWORD 7 @bit 8
//     Standard Inputs/MAIN.R2.In_From_HW/BYTE_[31] <-> Module 3 (Default IO)/Std. In (64 Bytes)/Input DWORD 7 @bit 16
//     Standard Inputs/MAIN.R2.In_From_HW/BYTE_[32] <-> Module 3 (Default IO)/Std. In (64 Bytes)/Input DWORD 7 @bit 24
//     Standard Inputs/MAIN.R2.In_From_HW/BYTE_[34] <-> Module 3 (Default IO)/Std. In (64 Bytes)/Input DWORD 8 @bit 8
//     Standard Inputs/MAIN.R2.In_From_HW/BYTE_[35] <-> Module 3 (Default IO)/Std. In (64 Bytes)/Input DWORD 8 @bit 16
//     Standard Inputs/MAIN.R2.In_From_HW/BYTE_[36] <-> Module 3 (Default IO)/Std. In (64 Bytes)/Input DWORD 8 @bit 24
//     Standard Inputs/MAIN.R2.In_From_HW/BYTE_[38] <-> Module 3 (Default IO)/Std. In (64 Bytes)/Input DWORD 9 @bit 8
//     Standard Inputs/MAIN.R2.In_From_HW/BYTE_[39] <-> Module 3 (Default IO)/Std. In (64 Bytes)/Input DWORD 9 @bit 16
//     Standard Inputs/MAIN.R2.In_From_HW/BYTE_[3] <-> Module 3 (Default IO)/Std. In (64 Bytes)/Input DWORD 0 @bit 16
//     Standard Inputs/MAIN.R2.In_From_HW/BYTE_[40] <-> Module 3 (Default IO)/Std. In (64 Bytes)/Input DWORD 9 @bit 24
//     Standard Inputs/MAIN.R2.In_From_HW/BYTE_[42] <-> Module 3 (Default IO)/Std. In (64 Bytes)/Input DWORD 10 @bit 8
//     Standard Inputs/MAIN.R2.In_From_HW/BYTE_[43] <-> Module 3 (Default IO)/Std. In (64 Bytes)/Input DWORD 10 @bit 16
//     Standard Inputs/MAIN.R2.In_From_HW/BYTE_[44] <-> Module 3 (Default IO)/Std. In (64 Bytes)/Input DWORD 10 @bit 24
//     Standard Inputs/MAIN.R2.In_From_HW/BYTE_[46] <-> Module 3 (Default IO)/Std. In (64 Bytes)/Input DWORD 11 @bit 8
//     Standard Inputs/MAIN.R2.In_From_HW/BYTE_[47] <-> Module 3 (Default IO)/Std. In (64 Bytes)/Input DWORD 11 @bit 16
//     Standard Inputs/MAIN.R2.In_From_HW/BYTE_[48] <-> Module 3 (Default IO)/Std. In (64 Bytes)/Input DWORD 11 @bit 24
//     Standard Inputs/MAIN.R2.In_From_HW/BYTE_[4] <-> Module 3 (Default IO)/Std. In (64 Bytes)/Input DWORD 0 @bit 24
//     Standard Inputs/MAIN.R2.In_From_HW/BYTE_[50] <-> Module 3 (Default IO)/Std. In (64 Bytes)/Input DWORD 12 @bit 8
//     Standard Inputs/MAIN.R2.In_From_HW/BYTE_[51] <-> Module 3 (Default IO)/Std. In (64 Bytes)/Input DWORD 12 @bit 16
//     Standard Inputs/MAIN.R2.In_From_HW/BYTE_[52] <-> Module 3 (Default IO)/Std. In (64 Bytes)/Input DWORD 12 @bit 24
//     Standard Inputs/MAIN.R2.In_From_HW/BYTE_[54] <-> Module 3 (Default IO)/Std. In (64 Bytes)/Input DWORD 13 @bit 8
//     Standard Inputs/MAIN.R2.In_From_HW/BYTE_[55] <-> Module 3 (Default IO)/Std. In (64 Bytes)/Input DWORD 13 @bit 16
//     Standard Inputs/MAIN.R2.In_From_HW/BYTE_[56] <-> Module 3 (Default IO)/Std. In (64 Bytes)/Input DWORD 13 @bit 24
//     Standard Inputs/MAIN.R2.In_From_HW/BYTE_[58] <-> Module 3 (Default IO)/Std. In (64 Bytes)/Input DWORD 14 @bit 8
